END_VAR
GVL_InstruTestUIVars.g_curTestCycles:=m_testCycles;
instruTestMode(i_slaveArm);
(*
IF ABS( m_targetGripAngLast-m_targetGripAng)>0.0001  THEN
  IF  m_targetGripAngLast-m_targetGripAng<0.0001   THEN
	  m_targetGripAng:=m_targetGripAng+m_openAngleInitCompensation*g_deg2rad;
  ELSE
	  m_targetGripAng:=m_targetGripAng;
  END_IF                       
END_IF
m_targetGripAngLast:=m_targetGripAng;
*)
//TIME
fbTime.timer(bStart:=TRUE,uiTimeHour=>GVL_InstruTestUIVars.g_testTimeHour,
						  uiTimeMinute=>GVL_InstruTestUIVars.g_testTimeMinute,
						  uiTimeSecond=>GVL_InstruTestUIVars.g_testTimeSecond);
// run OTG
FOR i:=1 TO 3  DO
	m_DHJntOTG[i].run(m_targetDHJntPos[i],0.0, o_cmdAcc=>,o_cmdVel=>m_cmdDHJntVel[i],o_cmdPos=> m_cmdDHJntPos[i+3]);
END_FOR
m_gripAngleOTG.run(m_targetGripAng,0.0, o_cmdAcc=>,o_cmdVel=>,o_cmdPos=>m_cmdGripAng);

// calculate target motor joint position from DH joint position
i_slaveArm.instrument.instruIK(m_cmdDHJntPos,m_cmdGripAng, o_jntPos=>m_cmdJntPos);

// command velocity
vecSub(m_cmdJntPos, m_lastCmdJntPos, m_cmdJntVel);
vecSelfMultiNum(m_cmdJntVel, g_slaveArmCtrlFreq);
m_lastCmdJntPos:=m_cmdJntPos;
END_METHOD

// override this function in each exact controller
METHOD PROTECTED calcCmdJntTrq : BOOL
VAR_IN_OUT CONSTANT
	i_endoscopePose : ST_Frame;
	i_masterStatus :ST_MasterStatus;
	i_setupStatus: ST_SetupStatus;
	i_slaveArm :FB_SlaveArm;
END_VAR

VAR 
	nullspaceMat :Mat7d;
	ctrlTrq : Vec7d;
	i : int ;
END_VAR
// set joint torque to zero in default
m_cmdJntTrq := g_zeroVec8d;

// instrument joint control
FOR i:=1 TO 5 DO 
	m_instruCmdJntPos[i]:=m_cmdJntPos[i+3];
	m_instruCmdJntVel[i]:=m_cmdJntVel[i+3];
END_FOR

IF i_slaveArm.instrument.instruType = InstruType_UltrasoundKnifeS OR i_slaveArm.instrument.instruType = InstruType_UltrasoundKnifeU THEN
	m_usKnifeController.run(m_instruCmdJntPos,m_instruCmdJntVel, m_targetGripForceLevel, i_slaveArm, o_cmdJntTrq=>m_instruCmdJntTrq);
ELSE
	m_instruController.run(m_instruCmdJntPos,m_instruCmdJntVel, m_cmdDHJntPos[6], m_cmdDHJntVel[6], m_targetGripForceLevel, i_slaveArm, o_cmdJntTrq=>m_instruCmdJntTrq);
END_IF

FOR i:=1 TO 5 DO
	m_cmdJntTrq[i+3]:=m_instruCmdJntTrq[i];
END_FOR
END_METHOD

METHOD PUBLIC init : BOOL
VAR_IN_OUT CONSTANT
	i_slaveArm	:FB_SlaveArm;
END_VAR
VAR_IN_OUT 
	r_slaveArmCtrlCmd :ST_SlaveArmCtrlCmds;
END_VAR

VAR
	i:int;
END_VAR
SUPER^.Init(i_slaveArm,r_slaveArmCtrlCmd);
m_lastCmdJntPos:=m_cmdJntPos;
m_jntOPMode[1] := DriverOPMode_PosTrq;
m_jntOPMode[2] := DriverOPMode_PosTrq;
m_jntOPMode[3] := DriverOPMode_PosTrq;
m_jntOPMode[4] := DriverOPMode_Trq;
m_jntOPMode[5] := DriverOPMode_Trq;
m_jntOPMode[6] := DriverOPMode_Trq;
m_jntOPMode[7] := DriverOPMode_Trq;
m_jntOPMode[8] := DriverOPMode_Trq;
m_armIdx:=i_slaveArm.armIdx;
fbTime.init();

//IF i_slaveArm.instrument.onChipData.m_InstruReadSucceed AND (InstruType_UltrasoundKnifeS = i_slaveArm.instrument.m_instruType 
 //  OR InstruType_UltrasoundKnifeU = i_slaveArm.instrument.m_instruType) THEN
    m_openAngleInitCompensation:=0;
	m_instruTestMode := 0;//GVL_InstruTestUIVars.g_testMode;
//ELSE
//	m_openAngleInitCompensation:=GVL_InstruTestUIVars.g_openAngleInitCompensation;
//	m_instruTestMode := GVL_InstruTestUIVars.g_testMode+10;
//END_IF
m_testStep := 0;
m_testCycles := 1;
m_cmdDHJntPos :=i_slaveArm.curDHJntPos;
m_cmdDHJntVel :=g_zeroVec6d;
m_targetGripAng := i_slaveArm.curGripAngle;
m_targetDHJntPos[1] := i_slaveArm.curDHJntPos[4];
m_targetDHJntPos[2] := i_slaveArm.curDHJntPos[5];
m_targetDHJntPos[3] := i_slaveArm.curDHJntPos[6];

// init instrument controller
m_instruController.init(i_slaveArm,m_maxGripCurrent,m_maxGripCtrlCurrent);
m_usKnifeController.init(i_slaveArm);
m_instruType := i_slaveArm.instrument.instruType;

FOR i:=1 TO 3  DO
	m_DHJntOTG[i].init(m_cmdDHJntPos[i+3], 0, m_maxJntVel[i], m_maxJntAcc[i], g_slaveArmCtrlCycleTime);
END_FOR

m_gripAngleOTG.init(m_targetGripAng, 0, m_maxJntVel[1], m_maxJntAcc[1], g_slaveArmCtrlCycleTime);
// update commands to arm
copyCmds(r_slaveArmCtrlCmd);


iStep:=5;
END_METHOD

PROPERTY InstruBacklash : Vec5d
GET
IF m_instruType = InstruType_UltrasoundKnifeS OR m_instruType = InstruType_UltrasoundKnifeU THEN
	instruBacklash := g_zeroVec5d;
ELSE
	instruBacklash := m_instruController.m_jntBacklash;
END_IF
END_GET
END_PROPERTY

METHOD instruTestMode : BOOL
VAR_IN_OUT CONSTANT
	i_slaveArm :FB_SlaveArm;
END_VAR
VAR
	i:INT;
END_VAR
CASE m_instruTestMode OF
	0:
		m_testStep := LIMIT(0,m_testStep, 12);
		m_instruPos:=m_postureTest;
		iStep1:=12;
		iStep2:=10;
	1:
		m_testStep := LIMIT(0,m_testStep, 8);
		m_instruPos:=m_openCloseTest;
		iStep1:=7;
		iStep2:=6;
	2:
		m_testStep := LIMIT(0,m_testStep, 59);
		m_instruPos:=m_openGripMoveTest;
		iStep1:=58;
		iStep2:=57;
	3:
		m_testStep := LIMIT(0,m_testStep, 59);
		m_instruPos:=m_openGripMoveTest;
		iStep1:=58;
		iStep2:=57;
	4:
		m_testStep := LIMIT(0,m_testStep, 28);
		m_instruPos:=m_openGripMoveTest;
		iStep1:=27;
		iStep2:=26;
	5:
		m_testStep := LIMIT(0,m_testStep, 25);
		m_instruPos:=m_openGripMoveTest;
		iStep1:=24;
		iStep2:=23;
	ELSE
		RETURN;
END_CASE
bstepMove:=TRUE;
IF iStep=15 OR iStep=0 THEN 
	GVL_InstruTestUIVars.g_inPos:=1;
ELSE
	GVL_InstruTestUIVars.g_inPos:=0;	
END_IF
GVL_InstruTestUIVars.m_postureTestStep:=m_testStep+1;
CASE iStep OF
	0:;
	5:  
		FOR i:=1 TO 3 BY 1 DO
			m_targetDHJntPos[i] := m_instruPos[m_testStep+1, i]*g_deg2rad;
		END_FOR
		m_targetGripAng := m_instruPos[m_testStep+1, 4]*g_deg2rad;
		m_targetGripForceLevel:=m_instruPos[m_testStep+1, 5];
		bstepMove:=FALSE;
		iStep:=10;
	10: 
		IF ABS(m_cmdDHJntPos[4]-m_targetDHJntPos[1])< g_jntCtrlAngTolLow 
		AND ABS(m_cmdDHJntPos[5]-m_targetDHJntPos[2])< g_jntCtrlAngTolLow 	
		AND ABS(m_cmdDHJntPos[6]-m_targetDHJntPos[3])< g_jntCtrlAngTolLow 
		AND ABS(m_cmdGripAng- m_targetGripAng)< g_jntCtrlAngTolLow 
		AND bstepMove  THEN
		    iStep:=15;
	    END_IF
	15: 
		IF  GVL_InstruTestUIVars.g_nextStep THEN
			m_testStep :=m_testStep + 1;
			iStep:=20;
		ELSIF  GVL_InstruTestUIVars.g_lastStep THEN
			IF m_testStep>=1 THEN
				m_testStep :=m_testStep - 1;
			ELSE
				IF m_testCycles>1 THEN
					m_testCycles:=m_testCycles-1	;
					m_testStep:=iStep1-1;
				END_IF
			END_IF
			iStep:=20;
		END_IF
		GVL_InstruTestUIVars.g_nextStep:=FALSE;
		GVL_InstruTestUIVars.g_lastStep:=FALSE;
	20:
		iStep:=5;
		IF m_testStep =iStep1 THEN
			m_testCycles:=m_testCycles+1;
			m_testStep := 0;
		END_IF

		IF m_testCycles>=2 THEN
			m_testCycles:=m_testCycles-1;
			iStep:=25;
		END_IF

	25: 
	    m_testStep:=iStep2+1;
		FOR i:=1 TO 3 BY 1 DO
			m_targetDHJntPos[i] := m_instruPos[m_testStep+1, i]*g_deg2rad;
		END_FOR
        m_targetGripAng := m_instruPos[m_testStep+1, 4]*g_deg2rad;
        m_targetGripForceLevel:=m_instruPos[m_testStep+1, 5];
		m_testStep:=iStep2+2;
		iStep:=30;
	
    30: IF ABS(m_cmdDHJntPos[4]-m_targetDHJntPos[1])< g_jntCtrlAngTolLow 
		AND ABS(m_cmdDHJntPos[5]-m_targetDHJntPos[2])< g_jntCtrlAngTolLow 
		AND ABS(m_cmdDHJntPos[6]-m_targetDHJntPos[3])< g_jntCtrlAngTolLow 
		AND ABS(m_cmdGripAng- m_targetGripAng)< g_jntCtrlAngTolLow THEN
		    iStep:=35;
	    END_IF
	35: 
	    m_isFinished := TRUE;
		iStep:=0;
END_CASE
END_METHOD

END_FUNCTION_BLOCK

// ---- FBs_SlaveControllers/FB_SlaveCtrlFrictionTest.TcPOU
// Brief: Slave Arm test
FUNCTION_BLOCK PUBLIC FB_SlaveCtrlFrictionTest EXTENDS FB_SlaveArmCtrlBase
VAR_INPUT
END_VAR
VAR_OUTPUT
END_VAR
VAR	
	m_jntOTG:ARRAY[1..6] OF FB_secOrdTrajFilter;
	m_testStep :INT:=0;
	m_cmdDHJntPos,m_targetDHJntPos :Vec6d;
	m_cmdDHJntAcc:Vec6d;
	m_cmdGripAng:LREAL:=0;
	m_lastCmdJntPos :Vec8d ;
	m_reachTargetPos:BOOL;
	m_currentRatioMotor2Jnt:LREAL;
	m_currentLoad1:LREAL := 50;
	m_currentLoad2:LREAL := 200;
	m_trqLoad1, m_trqLoad2 :LREAL;
	m_jntFrictionNum:Vec4d;
	
	m_jntFrictionNoLoad :Vec4d;
	m_jntFrictionWithLoad:Vec4d; 

	

	
//####################################################################

END_VAR

METHOD PROTECTED calcCmdJntPos : BOOL
VAR_IN_OUT CONSTANT
	i_endoscopePose : ST_Frame;
	i_masterStatus :ST_MasterStatus;
	i_setupStatus: ST_SetupStatus;
	i_slaveArm :FB_SlaveArm;
END_VAR

VAR 
	i:INT :=0;
	angErr:Vec6d;
	errThres :LREAL;
	jntVel:Vec8d;
	jntPos:Vec6d;
END_VAR
IF m_testStep > 8 THEN 
	m_isFinished := TRUE;
END_IF

m_jntOPMode := g_slaveAllPosTrqMode; 
m_cmdJntTrq :=g_zeroVec8d;
jntVel:=i_slaveArm.curJntVel;
jntPos:=i_slaveArm.curDHJntPos;
CASE m_testStep OF 
	0: // move to start posture
		m_targetDHJntPos[4]:=pi;
		m_targetDHJntPos[5]:=-PI/2;
		m_targetDHJntPos[6]:=-80*g_deg2rad;
	1: // yaw friction without load
		m_targetDHJntPos[4]:=pi;
		m_targetDHJntPos[5]:=-PI/2;
		m_targetDHJntPos[6]:=80*g_deg2rad;
		
		IF ABS(m_cmdDHJntAcc[6])<g_smallNum THEN
			m_jntFrictionNoLoad[1]:= (m_jntFrictionNoLoad[1]*m_jntFrictionNum[1]+ABS(i_slaveArm.filtJntCurrent[4]))/(m_jntFrictionNum[1]+1);
			m_jntFrictionNum[1]:=m_jntFrictionNum[1]+1;
			
			m_jntFrictionNoLoad[2]:= (m_jntFrictionNoLoad[2]*m_jntFrictionNum[2]+ABS(i_slaveArm.filtJntCurrent[5]))/(m_jntFrictionNum[2]+1);
			m_jntFrictionNum[2]:=m_jntFrictionNum[2]+1;
		END_IF
	2: // yaw finger1  friction with load 
		m_targetDHJntPos[4]:=pi;
		m_targetDHJntPos[5]:=-PI/2;
		m_targetDHJntPos[6]:=-80*g_deg2rad;
		m_jntOPMode[4]:= DriverOPMode_Trq;
		m_cmdJntTrq[4]:= m_trqLoad1;
		
		IF ABS(m_cmdDHJntAcc[6])<g_smallNum THEN
			m_jntFrictionWithLoad[2]:= (m_jntFrictionWithLoad[2]*m_jntFrictionNum[2]+ABS(i_slaveArm.filtJntCurrent[5]))/(m_jntFrictionNum[2]+1);
			m_jntFrictionNum[2]:=m_jntFrictionNum[2]+1;
		END_IF
	3: // yaw finger2  friction with load 
		m_targetDHJntPos[4]:=pi;
		m_targetDHJntPos[5]:=-PI/2;
		m_targetDHJntPos[6]:=80*g_deg2rad;
		m_jntOPMode[5]:= DriverOPMode_Trq;
		m_cmdJntTrq[5]:= m_trqLoad1;
		
		IF ABS(m_cmdDHJntAcc[6])<g_smallNum THEN
			m_jntFrictionWithLoad[1]:= (m_jntFrictionWithLoad[1]*m_jntFrictionNum[1]+ABS(i_slaveArm.filtJntCurrent[4]))/(m_jntFrictionNum[1]+1);
			m_jntFrictionNum[1]:=m_jntFrictionNum[1]+1;
		END_IF
		
	4: // pitch  friction without load 
		m_targetDHJntPos[4]:=pi;
		m_targetDHJntPos[5]:=-PI/2+75*g_deg2Rad;
		m_targetDHJntPos[6]:=0*g_deg2rad;
	5: 
		m_targetDHJntPos[4]:=pi;
		m_targetDHJntPos[5]:=-PI/2-75*g_deg2Rad;
		m_targetDHJntPos[6]:=0*g_deg2rad;
		
		IF ABS(m_cmdDHJntAcc[5])<g_smallNum THEN
			m_jntFrictionNoLoad[3]:= (m_jntFrictionNoLoad[3]*m_jntFrictionNum[3]+ABS(i_slaveArm.filtJntCurrent[6]))/(m_jntFrictionNum[3]+1);
			m_jntFrictionNum[3]:=m_jntFrictionNum[3]+1;
		END_IF
		
	6: // pitch  friction with load 
		m_targetDHJntPos[4]:=pi;
		m_targetDHJntPos[5]:=-PI/2+75*g_deg2Rad;
		m_targetDHJntPos[6]:=0*g_deg2rad;
		m_jntOPMode[4]:= DriverOPMode_Trq;
		m_cmdJntTrq[4]:= m_trqLoad2;
		m_jntOPMode[5]:= DriverOPMode_Trq;
		m_cmdJntTrq[5]:= m_trqLoad2;
		
		IF ABS(m_cmdDHJntAcc[5])<g_smallNum THEN
			m_jntFrictionWithLoad[3]:= (m_jntFrictionWithLoad[3]*m_jntFrictionNum[3]+ABS(i_slaveArm.filtJntCurrent[6]))/(m_jntFrictionNum[3]+1);
			m_jntFrictionNum[3]:=m_jntFrictionNum[3]+1;
		END_IF
	7: // roll friction without load 
		m_targetDHJntPos[4]:=-pi;
		m_targetDHJntPos[5]:=-PI/2+75*g_deg2Rad;
		m_targetDHJntPos[6]:=0*g_deg2rad;
		IF ABS(m_cmdDHJntAcc[4])<g_smallNum THEN
			m_jntFrictionNoLoad[4]:= (m_jntFrictionNoLoad[4]*m_jntFrictionNum[4]+ABS(i_slaveArm.filtJntCurrent[7]))/(m_jntFrictionNum[4]+1);
			m_jntFrictionNum[4]:=m_jntFrictionNum[4]+1;
		END_IF
	8: 
		m_targetDHJntPos[4]:=-pi;
		m_targetDHJntPos[5]:=-PI/2;
		m_targetDHJntPos[6]:=0*g_deg2rad;
		
END_CASE

// check if finish current motion
vecSub(m_cmdDHJntPos, m_targetDHJntPos, angErr);
IF norm(angErr)< 1*g_deg2Rad AND norm(jntVel)<1*g_deg2Rad THEN
	m_testStep := m_testStep+1;
	m_jntFrictionNum:=g_zeroVec4d;
END_IF


FOR i:=4 TO 6 DO 
	m_jntOTG[i].run(m_targetDHJntPos[i],0.0, o_cmdAcc=>m_cmdDHJntAcc[i],o_cmdVel=>,o_cmdPos=> m_cmdDHJntPos[i]);
END_FOR

i_slaveArm.instrument.instruIK(m_cmdDHJntPos,m_cmdGripAng, o_jntPos=>m_cmdJntPos);

// command velocity
vecSub(m_cmdJntPos, m_lastCmdJntPos, m_cmdJntVel);
vecSelfMultiNum(m_cmdJntVel, g_slaveArmCtrlFreq);
m_lastCmdJntPos:=m_cmdJntPos;
END_METHOD

// override this function in each exact controller
METHOD PROTECTED calcCmdJntTrq : BOOL
VAR_IN_OUT CONSTANT
	i_endoscopePose : ST_Frame;
	i_masterStatus :ST_MasterStatus;
	i_setupStatus: ST_SetupStatus;
	i_slaveArm :FB_SlaveArm;
END_VAR

VAR 
	nullspaceMat :Mat7d;
	ctrlTrq : Vec7d;
	i : int ;
END_VAR
END_METHOD

METHOD PUBLIC init : BOOL
VAR_IN_OUT CONSTANT
	i_slaveArm	:FB_SlaveArm;
END_VAR
VAR_IN_OUT 
	r_slaveArmCtrlCmd :ST_SlaveArmCtrlCmds;
END_VAR

VAR
	i:int;
END_VAR
SUPER^.Init(i_slaveArm,r_slaveArmCtrlCmd);
m_lastCmdJntPos:=m_cmdJntPos;
m_jntOPMode := g_slaveAllPosTrqMode; 

m_testStep:=0;
m_cmdDHJntPos :=i_slaveArm.curDHJntPos;
m_targetDHJntPos:=m_cmdDHJntPos;
m_cmdGripAng:=0;
m_lastCmdJntPos:=m_cmdJntPos;
m_reachTargetPos:=FALSE;

m_currentRatioMotor2Jnt:=GVL_SlaveMotorParameters.g_motorTrqConst[4]*GVL_SlaveMotorParameters.g_motorReduction[4]/1000;
m_trqLoad1 := m_currentLoad1 * m_currentRatioMotor2Jnt;
m_trqLoad2 := m_currentLoad2 * m_currentRatioMotor2Jnt;


FOR i:=1 TO 6  DO
	m_jntOTG[i].init(m_cmdDHJntPos[i], 0, 10*g_deg2Rad, 4, g_slaveArmCtrlCycleTime);
END_FOR

m_jntFrictionNoLoad:=g_zeroVec4d;
m_jntFrictionWithLoad:=g_zeroVec4d;
m_jntFrictionNum:=g_zeroVec4d;

// update commands to arm
copyCmds(r_slaveArmCtrlCmd);
END_METHOD

END_FUNCTION_BLOCK

// ---- FBs_SlaveControllers/FB_SlaveCtrMotorGoHome.TcPOU
// Brief: Mounting Panel
FUNCTION_BLOCK PUBLIC FB_SlaveCtrMotorGoHome EXTENDS FB_SlaveArmCtrlBase
VAR
	// motorGoHomeStatus
	m_motorGoHomeStatus :INT := 0;
	
	// mount motion planning
	m_jntOTG :ARRAY[1..5] OF FB_secOrdTrajFilter;
	m_motorGoHomeVel :LREAL := 2*pi;
	m_motorGoHomeAcc :LREAL := 4*pi;
	m_targetHomePos :Vec5d;
END_VAR

// override this function in each exact controller
METHOD PROTECTED calcCmdJntPos : BOOL
VAR_IN_OUT CONSTANT
	i_endoscopePose : ST_Frame;
	i_masterStatus :ST_MasterStatus;
	i_setupStatus: ST_SetupStatus;
	i_slaveArm :FB_SlaveArm;
END_VAR

VAR 
	i :INT;
	curJntPos :Vec8d;
	cycleNum :LREAL;
END_VAR

curJntPos := i_slaveArm.curJntPos;

CASE m_motorGoHomeStatus OF
	
	// determine zero position 
	0:
		FOR i:=1 TO 5 DO
			cycleNum := FLOOR(curJntPos[i+3]/g_2pi);
			m_targetHomePos[i]:=cycleNum* g_2Pi;
		END_FOR
		m_motorGoHomeStatus :=1;
	
	// move back to zero position
	1:
		m_isFinished:=TRUE;
		FOR i:=1 TO 5 DO
			IF ABS(m_targetHomePos[i]-curJntPos[i+3])>GVL_SlaveControlParameters.g_jntCtrlAngTolHigh THEN
				m_isFinished:=FALSE;
				EXIT;
			END_IF
		END_FOR
END_CASE


FOR i:=1 TO 5 DO
	m_jntOTG[i].run(m_targetHomePos[i],0.0, o_cmdAcc=>m_cmdJntAcc[3+i],o_cmdVel=>m_cmdJntVel[3+i],o_cmdPos=>m_cmdJntPos[i+3]);
END_FOR
END_METHOD

METHOD PUBLIC init : BOOL
VAR_IN_OUT CONSTANT
	i_slaveArm	:FB_SlaveArm;
END_VAR
VAR_IN_OUT 
	r_slaveArmCtrlCmd :ST_SlaveArmCtrlCmds;
END_VAR
VAR
	i : INT;
END_VAR
SUPER^.Init(i_slaveArm,r_slaveArmCtrlCmd);//T
m_jntOPMode[4] := DriverOPMode_Pos;
m_jntOPMode[5] := DriverOPMode_Pos;
m_jntOPMode[6] := DriverOPMode_Pos;
m_jntOPMode[7] := DriverOPMode_Pos;
m_jntOPMode[8] := DriverOPMode_Pos;

m_motorGoHomeStatus:=0;
FOR i:=1 TO 5 DO
	m_targetHomePos[i]:=m_cmdJntPos[i+3];
	m_jntOTG[i].init(m_targetHomePos[i], 0,m_motorGoHomeVel, m_motorGoHomeAcc, g_slaveArmCtrlCycleTime);
END_FOR

// update commands to arm
copyCmds(r_slaveArmCtrlCmd);
END_METHOD

END_FUNCTION_BLOCK

// ---- FBs_Robots/FB_SlaveRobot.TcPOU
FUNCTION_BLOCK FB_SlaveRobot
VAR
	// slave arms, responsible for arm kinematic and control
	m_slaveArms :ARRAY[1..g_sArmNum] OF FB_SlaveArm;
	
	// arm light control word
	m_lightCrlWord :ARRAY [1..4] OF UDINT;
	
	// arm state
	m_slaveArmState:ARRAY[1..g_sArmNum] OF E_SlaveArmState:=[g_sArmNum(E_SlaveArmState.SlaveArmState_Error)];
	m_lastSlaveArmState:ARRAY[1..g_sArmNum] OF E_SlaveArmState:=[g_sArmNum(E_SlaveArmState.SlaveArmState_Error)];
	m_nextSlaveArmState:ARRAY[1..g_sArmNum] OF E_SlaveArmState:=[g_sArmNum(E_SlaveArmState.SlaveArmState_Error)];
	
	// flag if panel and instrument mounted
	m_panelMountedFlag :ARRAY[1..g_sArmNum] OF BOOL :=[g_sArmNum(FALSE)];
	m_instrumentMountedFlag :ARRAY[1..g_sArmNum] OF BOOL :=[g_sArmNum(FALSE)];
	
	// all arm controller instance 
	m_armCtrlFactory :ARRAY[1..g_sArmNum,1..SlaveArmState_totalNum] OF I_SlaveArmCtrl;
	m_armError :ARRAY[1..g_sArmNum] OF FB_SlaveCtrlError;
	m_armInit :ARRAY[1..g_sArmNum] OF FB_SlaveCtrlInit;
	m_armSelfCheck :ARRAY[1..g_sArmNum] OF FB_SlaveCtrlSelfCheck;
	m_armStandBy :ARRAY[1..g_sArmNum] OF FB_SlaveCtrlStandBy;
	m_mountPanel :ARRAY[1..g_sArmNum] OF FB_SlaveCtrlMountPanel;
	m_panelReady :ARRAY[1..g_sArmNum] OF FB_SlaveCtrlPanelReady;
	m_mountInstru :ARRAY[1..g_sArmNum] OF FB_SlaveCtrlMountInstru;
	m_instruReady :ARRAY[1..g_sArmNum] OF FB_SlaveCtrlInstruReady;
	m_armMasterSlave :ARRAY[1..g_sArmNum] OF FB_SlaveCtrlMasterSlave;
	m_scopeReady :ARRAY[1..g_sArmNum] OF FB_SlaveCtrlScopeReady;
	m_armEndoscope :ARRAY[1..g_sArmNum] OF FB_SlaveCtrlEndoscope;
	m_armAdjust :ARRAY[1..g_sArmNum] OF FB_SlaveCtrlAdjust;
	m_armPackage :ARRAY[1..g_sArmNum] OF FB_SlaveCtrlPackage;
	m_armCart :ARRAY[1..g_sArmNum] OF FB_SlaveCtrlCart;
	m_armGraCali :ARRAY[1..g_sArmNum] OF FB_SlaveCtrlGraCali;
	m_armTest :ARRAY[1..g_sArmNum] OF FB_SlaveCtrlTest;
	m_instruRetract :ARRAY[1..g_sArmNum] OF FB_SlaveCtrlInstruRetract;
	m_instruInvasion :ARRAY[1..g_sArmNum] OF FB_SlaveCtrlInstruInvasion;
	m_armDisable :ARRAY[1..g_sArmNum] OF FB_SlaveCtrlDisable;
	m_instruCali :ARRAY[1..g_sArmNum] OF FB_SlaveCtrlInstruCali;
	m_scopeToggle :ARRAY[1..g_sArmNum] OF FB_SlaveCtrlScopeToggle;
	m_Performance :ARRAY[1..g_sArmNum] OF FB_SlaveCtrlPerformance;
	m_armStop :ARRAY[1..g_sArmNum] OF FB_SlaveCtrlStop;
	m_instruAutoTest :ARRAY[1..g_sArmNum] OF FB_SlaveCtrlInstruAutoTest;
	m_instruManualTest :ARRAY[1..g_sArmNum] OF FB_SlaveCtrlInstruManualTest;
	m_instruVerify :ARRAY[1..g_sArmNum] OF FB_SlaveCtrlInstruVerify;
	m_frictionTest :ARRAY[1..g_sArmNum] OF FB_SlaveCtrlFrictionTest;
	
	// arm controller interface
	m_armCtrl :ARRAY[1..g_sArmNum] OF I_SlaveArmCtrl;
	m_armCtrlCmds :ARRAY[1..g_sArmNum] OF ST_SlaveArmCtrlCmds;
	m_motorGoHome: ARRAY[1..g_sArmNum] OF FB_SlaveCtrMotorGoHome;
	m_powerBoxCalibration: ARRAY[1..g_sArmNum] OF FB_SlaveCtrlPowerBoxCalibration;
	fbTonMotorGoHomeState: TON;
	fbTonPowerBoxCalibrationState: TON;
	m_endoscopeTest: ARRAY[1..g_sArmNum] OF FB_SlaveCtrlInstruEndoscopeTest;
	m_enableMode:BOOL;
	
	m_frictionTestButtonRise :R_TRIG;
	m_frictionTestButtonFall :F_TRIG;
	m_frictionTestStart, m_frictionTestEnd:BOOL;
END_VAR

METHOD PROTECTED controllerTransit : BOOL
VAR_INPUT
END_VAR
VAR
	i:int;
END_VAR
FOR i:=1 TO g_sArmNum DO 
	// Controller transit
	IF m_nextSlaveArmState[i]<> m_slaveArmState[i] THEN
		// reset current controller
		m_armCtrl[i].reset();
		
		// transit to new controller
		m_lastSlaveArmState[i]:=m_slaveArmState[i];
		m_slaveArmState[i]:=m_nextSlaveArmState[i];
		m_armCtrl[i]:=m_armCtrlFactory[i,m_slaveArmState[i]];
		
		// init next controller
		m_armCtrl[i].Init(m_slaveArms[i],m_armCtrlCmds[i]);
		m_slaveArms[i].updateCmds(m_armCtrlCmds[i]);
	END_IF
END_FOR
END_METHOD

METHOD PUBLIC Init : BOOL
VAR_INPUT
END_VAR
VAR
	i:INT;
END_VAR
FOR i:=1 TO g_sArmNum DO
	// arm init
	m_slaveArms[i].Init(i);
	m_slaveArmState[i]:=SlaveArmState_Init;
	m_lastSlaveArmState[i]:=SlaveArmState_Init;
	m_nextSlaveArmState[i]:=SlaveArmState_Init;
	
	// command init
	m_armCtrlCmds[i].m_jntEnableFlag := g_zeroVec8i;
	m_armCtrlCmds[i].m_jntOPMode := g_slaveAllPosMode;
	m_armCtrlCmds[i].m_cmdCartPose := m_slaveArms[i].curCartPose;
	m_armCtrlCmds[i].m_cmdCartTwist := g_zeroVec6d;
	m_armCtrlCmds[i].m_cmdJntPos := m_slaveArms[i].curJntPos;
	m_armCtrlCmds[i].m_cmdJntVel := g_zeroVec8d;
	m_armCtrlCmds[i].m_cmdJntAcc := g_zeroVec8d;
	m_armCtrlCmds[i].m_cmdJntTrq := g_zeroVec8d;
	
	// generate controller factory
	m_armCtrlFactory[i,SlaveArmState_Error] := m_armError[i];
	m_armCtrlFactory[i,SlaveArmState_Init] := m_armInit[i];
	m_armCtrlFactory[i,SlaveArmState_SelfCheck] := m_armSelfCheck[i];
	m_armCtrlFactory[i,SlaveArmState_Standby] := m_armStandBy[i];
	m_armCtrlFactory[i,SlaveArmState_MountPanel] := m_mountPanel[i];
	m_armCtrlFactory[i,SlaveArmState_PanelReady] := m_panelReady[i];
	m_armCtrlFactory[i,SlaveArmState_MountInstru] := m_mountInstru[i];
	m_armCtrlFactory[i,SlaveArmState_InstruReady] := m_instruReady[i];
	m_armCtrlFactory[i,SlaveArmState_MasterSlave] := m_armMasterSlave[i];
	m_armCtrlFactory[i,SlaveArmState_ScopeReady] := m_scopeReady[i];
	m_armCtrlFactory[i,SlaveArmState_EndoScope] := m_armEndoscope[i];
	m_armCtrlFactory[i,SlaveArmState_Adjust] := m_armAdjust[i];
	m_armCtrlFactory[i,SlaveArmState_Package] := m_armPackage[i];
	m_armCtrlFactory[i,SlaveArmState_Cart] := m_armCart[i];
	m_armCtrlFactory[i,SlaveArmState_GravityCali] := m_armGraCali[i];
	m_armCtrlFactory[i,SlaveArmState_Test] := m_armTest[i];
	m_armCtrlFactory[i,SlaveArmState_InstruRetract] := m_instruRetract[i];
	m_armCtrlFactory[i,SlaveArmState_InstruInvasion] := m_instruInvasion[i];
	m_armCtrlFactory[i,SlaveArmState_Disable] := m_armDisable[i];
	m_armCtrlFactory[i,SlaveArmState_InstruCali] := m_instruCali[i];
	m_armCtrlFactory[i,SlaveArmState_ScopeToggle] := m_scopeToggle[i];
	m_armCtrlFactory[i,SlaveArmState_Performance] := m_Performance[i];
	m_armCtrlFactory[i,SlaveArmState_Stop] := m_armStop[i];
	m_armCtrlFactory[i,SlaveArmState_InstruAutoTest] := m_instruAutoTest[i];
	m_armCtrlFactory[i,SlaveArmState_InstruManualTest] := m_instruManualTest[i];
	m_armCtrlFactory[i,SlaveArmState_InstruVerify] := m_instruVerify[i];
	m_armCtrlFactory[i,SlaveArmState_MotorGoHome] := m_motorGoHome[i];
	m_armCtrlFactory[i,SlaveArmState_PowerBoxCalibration] := m_powerBoxCalibration[i];
	m_armCtrlFactory[i,SlaveArmState_EndoscopeTest] := m_endoscopeTest[i];
	m_armCtrlFactory[i,SlaveArmState_FrictionTest] := m_frictionTest[i];
	// assign controller
	m_armCtrl[i]:=m_armCtrlFactory[i,m_slaveArmState[i]];
	m_armCtrl[i].Init(m_slaveArms[i],m_armCtrlCmds[i]);
END_FOR
END_METHOD

METHOD PUBLIC run : BOOL
VAR_IN_OUT CONSTANT
	i_slaveInputDataPool:ST_SlaveInputDataPool;
END_VAR
VAR
	i:INT;
	nullScopePose :ST_Frame;
	nullSetupStatus:ST_SetupStatus;
	nullMasterStatus:ST_MasterStatus;
	
	
END_VAR
FOR i:=1 TO g_sArmNum DO
	// update dynamic data
	m_slaveArms[i].updateDyna(i_slaveInputDataPool.m_slaveDynaData);
								
	// update slave arm kinematics
	m_slaveArms[i].updateStatus();
END_FOR

//update arm light
updateArmLight(i_slaveInputDataPool);

// state machine transition
stateMachine(i_slaveInputDataPool);

// controller transition
controllerTransit();

FOR i:=1 TO g_sArmNum DO
	// null ptr check
	ASSERT(0 <> m_armCtrl[i]);
	
	// run controller
	m_armCtrl[i].run(nullScopePose, nullMasterStatus, nullSetupStatus,m_SlaveArms[i],m_armCtrlCmds[i]);

	// update commands to drivers
	m_slaveArms[i].updateCmds(m_armCtrlCmds[i]);

END_FOR
// ################# update insrument UI data #########################################
FOR i:=1 TO 5 DO 
	GVL_InstruTestUIVars.g_curInstruJntPos[i]:= m_slaveArms[1].curJntPos[i+3];
	GVL_InstruTestUIVars.g_curInstruJntCurrent[i]:= m_slaveArms[1].filtJntCurrent[i+3];
	GVL_InstruTestUIVars.g_instruZeroPos[i]:= m_slaveArms[1].instrument.onChipData.m_InstruPos[i];
END_FOR

FOR i:=1 TO 3 DO
		GVL_InstruTestUIVars.g_curInstruDHPos[i]:= m_slaveArms[1].curDHJntPos[i+3];
END_FOR

GVL_InstruTestUIVars.g_curGripAng := m_slaveArms[1].curGripAngle;
GVL_InstruTestUIVars.g_enabled := m_slaveArms[1].m_joints[6].isEnabled() ;

m_frictionTestButtonRise(CLK:=GVL_InstruTestUIVars.g_instruFrictionTest,  Q=>m_frictionTestStart);
m_frictionTestButtonFall(CLK:=GVL_InstruTestUIVars.g_instruFrictionTest,  Q=>m_frictionTestEnd);
END_METHOD

// state machine check and transit 
METHOD PROTECTED stateMachine : BOOL
VAR_IN_OUT CONSTANT
		i_slavesInputDataPool:ST_SlaveInputDataPool;
END_VAR
VAR
	i,j:INT;
END_VAR
// check instrument state
FOR i:=1 TO g_sArmNum DO
	// statues check
	IF m_slaveArms[i].panelOn = FALSE THEN
		m_panelMountedFlag[i]:=FALSE;
	END_IF
	IF m_slaveArms[i].instruOn = FALSE THEN
		m_instrumentMountedFlag[i]:=FALSE;
	END_IF
END_FOR

// state machine transit
FOR i:=1 TO g_sArmNum DO
	CASE m_slaveArmState[i] OF
		// init
		SlaveArmState_Init:
			m_slaveArms[i].instrument.resetArmLED :=TRUE;
			// to standby
			IF m_armCtrl[i].isFinished  THEN
				m_nextSlaveArmState[i]:=SlaveArmState_Standby;
			END_IF
		
		//standby
		SlaveArmState_Standby:
			// to mount panel
			IF m_slaveArms[i].panelOn AND ((GVL_InstruTestUIVars.g_snappingSeparator AND NOT m_slaveArms[i].instruOn) OR  m_panelMountedFlag[i] )AND NOT GVL_InstruTestUIVars.g_powerBoxCalibration THEN 
				IF m_panelMountedFlag[i] THEN
					m_nextSlaveArmState[i]:=SlaveArmState_PanelReady;
				ELSE
					m_nextSlaveArmState[i]:=SlaveArmState_MountPanel;
				END_IF
			ELSIF GVL_InstruTestUIVars.g_goHome AND NOT m_slaveArms[i].instruOn THEN  
				GVL_InstruTestUIVars.g_beHomed:=FALSE;
				m_nextSlaveArmState[i]:=SlaveArmState_MotorGoHome;
			END_IF
			IF GVL_InstruTestUIVars.g_powerBoxCalibration THEN
				GVL_InstruTestUIVars.g_powerBoxCalibrationed:=FALSE;;
				IF m_slaveArms[i].panelOn THEN 
					m_nextSlaveArmState[i]:=SlaveArmState_PowerBoxCalibration;
				END_IF
			END_IF
		SlaveArmState_MotorGoHome:
			// to Standby
			IF m_armCtrl[i]. isFinished THEN
				m_nextSlaveArmState[i]:=SlaveArmState_Standby;
				GVL_InstruTestUIVars.g_beHomed:=TRUE;
			// to standby
			ELSIF fbTonMotorGoHomeState.Q THEN
				m_nextSlaveArmState[i]:=SlaveArmState_Standby;
			END_IF
		SlaveArmState_PowerBoxCalibration:
			IF m_armCtrl[i]. isFinished THEN
				GVL_InstruTestUIVars.g_powerBoxCalibration:=FALSE;
				GVL_InstruTestUIVars.g_powerBoxCalibrationed:=TRUE;
				FOR j:=4 TO g_sJntNum DO
					GVL_InstruTestUIVars.g_powerBoxCalibrationPos[i,j]:=SlaveArmControl.m_slaveRobot.m_slaveArms[i].m_joints[j].m_motorInputs.m_linkEncoder;
				END_FOR
				GVL_SlaveJointEncoderCaliData.g_caliLinkEncoder:=GVL_InstruTestUIVars.g_powerBoxCalibrationPos;
				IF NOT m_slaveArms[i].panelOn THEN
					GVL_InstruTestUIVars.g_powerBoxCalibrationFlag:=FALSE;
					m_nextSlaveArmState[i]:=SlaveArmState_Standby;;
					m_slaveArms[i].setSaveCaliLinkEncoder();
				END_IF
			// to standby
			ELSIF fbTonPowerBoxCalibrationState.Q AND NOT m_slaveArms[i].panelOn THEN
				m_nextSlaveArmState[i]:=SlaveArmState_Standby;
			END_IF
		//mount panel
		SlaveArmState_MountPanel:
			// to panel ready
			IF m_armCtrl[i]. isFinished THEN
				m_nextSlaveArmState[i]:=SlaveArmState_PanelReady;
				m_panelMountedFlag[i] :=TRUE;
				
			// to standby
			ELSIF NOT(m_slaveArms[i].panelOn) THEN
				m_nextSlaveArmState[i]:=SlaveArmState_Standby;
			END_IF
		
		//panel ready
		SlaveArmState_PanelReady:
			// to standby
			IF NOT(m_slaveArms[i].panelOn) THEN
				m_nextSlaveArmState[i]:=SlaveArmState_Standby;
			
			// to instrument caliberation
			ELSIF GVL_InstruTestUIVars.g_instruCaliFlag THEN
				m_nextSlaveArmState[i] := SlaveArmState_InstruCali;
			ELSIF (GVL_InstruTestUIVars.g_instrumentAutoSnapping OR m_instrumentMountedFlag[i]) AND m_slaveArms[i].instruOn   THEN
				IF m_instrumentMountedFlag[i] THEN
					// to scope ready
					IF  InstruType_endoscope = m_slaveArms[i].instrument.m_instruType AND m_slaveArms[i].instruReady() THEN 
						m_nextSlaveArmState[i]:=SlaveArmState_ScopeReady;
					// to instrument ready
					ELSE
						m_nextSlaveArmState[i]:=SlaveArmState_InstruReady;
					END_IF
				// to mount instrument/endoscope
				ELSE
					m_nextSlaveArmState[i]:=SlaveArmState_MountInstru;
				END_IF
			END_IF
			
		//mount instrument
		SlaveArmState_MountInstru:
			// to panel ready
			IF NOT(m_slaveArms[i].instruOn)  THEN
				m_nextSlaveArmState[i]:=SlaveArmState_PanelReady;
			ELSIF m_armCtrl[i].isFinished THEN
				m_instrumentMountedFlag[i] :=TRUE;
				m_nextSlaveArmState[i]:=SlaveArmState_PanelReady;
				
			END_IF
		
		// instrument ready
		SlaveArmState_InstruReady:
			// to instrument standby
			IF  NOT(m_slaveArms[i].instruOn)  THEN
				m_nextSlaveArmState[i]:=SlaveArmState_Standby;
				GVL_InstruTestUIVars.g_readRFIDFlag:=FALSE;
			// to instrument caliberation
			ELSIF GVL_InstruTestUIVars.g_instruCaliFlag THEN
				m_nextSlaveArmState[i] := SlaveArmState_InstruCali;
				
			// to instrument auto test
			ELSIF GVL_InstruTestUIVars.g_instruAutoTestFlag THEN
				m_nextSlaveArmState[i] := SlaveArmState_InstruAutoTest;
				
			// to instrument manual test
			ELSIF GVL_InstruTestUIVars.g_instruManualTestFlag THEN
				m_nextSlaveArmState[i] := SlaveArmState_InstruManualTest;
				
			// to instrument verify
			ELSIF GVL_InstruTestUIVars.g_instruVerifyFlag THEN
				m_nextSlaveArmState[i] := SlaveArmState_InstruVerify;
				
			// to instrument verify
			ELSIF GVL_InstruTestUIVars.g_endoscopeTest THEN
				m_nextSlaveArmState[i] := SlaveArmState_EndoscopeTest;
				
			//to friction Test
			ELSIF m_frictionTestStart THEN
				m_nextSlaveArmState[i] := SlaveArmState_FrictionTest;
			END_IF
			
		//instrument caliberation
		SlaveArmState_InstruCali:
			// to standby
			IF  NOT(GVL_InstruTestUIVars.g_instruCaliFlag)  THEN
				m_nextSlaveArmState[i]:=SlaveArmState_Standby;
			END_IF
			
		//instrument auto test
		SlaveArmState_InstruAutoTest:
			// to stop
			IF  NOT( m_slaveArms[1].instruOn) OR NOT(GVL_InstruTestUIVars.g_instruAutoTestFlag)  THEN
				m_nextSlaveArmState[i]:=SlaveArmState_Stop;
				GVL_InstruTestUIVars.g_readRFIDFlag:=FALSE;
				m_armStop[i].setInstruBacklash(m_instruAutoTest[i].InstruBacklash);
			END_IF
			IF m_armCtrl[i].isFinished THEN
				GVL_InstruTestUIVars.g_instruAutoTestFlag:=FALSE;
			END_IF
		//instrument manual test
		SlaveArmState_InstruManualTest:
			// to stop
			IF  NOT( m_slaveArms[1].instruOn) OR NOT(GVL_InstruTestUIVars.g_instruManualTestFlag)  THEN
				m_nextSlaveArmState[i]:=SlaveArmState_Stop;
				m_armStop[i].setInstruBacklash(m_instruManualTest[i].InstruBacklash);
				GVL_InstruTestUIVars.g_readRFIDFlag:=FALSE;
			END_IF
			
		//instrument verify
		SlaveArmState_InstruVerify:
			// to stop
			IF  NOT( m_slaveArms[1].instruOn) OR NOT(GVL_InstruTestUIVars.g_instruVerifyFlag)  THEN
				m_nextSlaveArmState[i]:=SlaveArmState_Stop;
				GVL_InstruTestUIVars.g_readRFIDFlag:=FALSE;
				m_armStop[i].setInstruBacklash(m_instruVerify[i].InstruBacklash);
			END_IF
			IF m_armCtrl[i].isFinished THEN
				GVL_InstruTestUIVars.g_instruVerifyFlag:=FALSE;
			END_IF
			
		//arm stop
		SlaveArmState_Stop:
			// to standby
			IF  m_armCtrl[i].isFinished THEN
				m_nextSlaveArmState[i]:=SlaveArmState_Standby;
			END_IF
			
		SlaveArmState_Disable:
			// to init
			IF  NOT GVL_InstruTestUIVars.g_powerOn  THEN
				m_nextSlaveArmState[i]:=SlaveArmState_Init;
			END_IF
		    IF  NOT( m_slaveArms[1].instruOn) THEN
				m_nextSlaveArmState[i]:=SlaveArmState_Init;
			END_IF
			
		SlaveArmState_EndoscopeTest:
			IF  NOT( m_slaveArms[1].instruOn) OR NOT(GVL_InstruTestUIVars.g_endoscopeTest)  THEN
				m_nextSlaveArmState[i]:=SlaveArmState_Stop;
			END_IF
			
		SlaveArmState_FrictionTest:
			// to stop
			IF  NOT( m_slaveArms[1].instruOn) OR m_armCtrl[i].isFinished OR m_frictionTestEnd  THEN
				m_nextSlaveArmState[i]:=SlaveArmState_Standby;
			END_IF
	END_CASE
	IF NOT m_slaveArms[i].instruOn THEN
		GVL_InstruTestUIVars.g_instruCaliState:=FALSE;
	END_IF
	IF GVL_InstruTestUIVars.g_powerOn THEN 
		m_nextSlaveArmState[i]:=SlaveArmState_Disable;
	END_IF
	IF GVL_InstruTestUIVars.g_motorStops THEN 
		GVL_InstruTestUIVars.g_motorStops:=FALSE;
		m_nextSlaveArmState[i]:=SlaveArmState_Stop;
	END_IF
	IF m_slaveArmState[i]<>SlaveArmState_PowerBoxCalibration AND m_slaveArmState[i]<>SlaveArmState_Standby THEN
		GVL_InstruTestUIVars.g_powerBoxCalibration:=FALSE;
	END_IF
	IF m_slaveArmState[i]<>SlaveArmState_MotorGoHome AND m_slaveArmState[i]<>SlaveArmState_Standby THEN
		GVL_InstruTestUIVars.g_beHomed:=FALSE;
	END_IF
	
	
GVL_InstruTestUIVars.g_stateMachine:=m_slaveArmState[i];
	IF GVL_InstruTestUIVars.g_manualPowerBoxCalibration THEN
		FOR j:=4 TO g_sJntNum DO
			GVL_InstruTestUIVars.g_powerBoxCalibrationPos[i,j]:=SlaveArmControl.m_slaveRobot.m_slaveArms[i].m_joints[j].m_motorInputs.m_linkEncoder;
		END_FOR
		//GVL_SlaveJointEncoderCaliData.g_caliLinkEncoder:=GVL_InstruTestUIVars.g_powerBoxCalibrationPos;
		GVL_InstruTestUIVars.g_manualPowerBoxCalibration:=FALSE;
		GVL_InstruTestUIVars.g_powerBoxCalibrationFlag:=FALSE;
		m_slaveArms[i].setSaveCaliLinkEncoder();
	END_IF
END_FOR


m_enableMode:=TRUE;
GVL_InstruTestUIVars.g_logOutEnable:=GVL_InstruTestUIVars.g_stateMachine<>SlaveArmState_InstruAutoTest;
GVL_InstruTestUIVars.g_snappingSeparatoring:=GVL_InstruTestUIVars.g_stateMachine=SlaveArmState_MountPanel;
GVL_InstruTestUIVars.g_instruAutoSnapping:=GVL_InstruTestUIVars.g_stateMachine=SlaveArmState_MountInstru;
GVL_InstruTestUIVars.g_instruCalibrationing:=m_instruCali[1].getState AND GVL_InstruTestUIVars.g_stateMachine=SlaveArmState_InstruCali;
GVL_MES.g_autoTestMode:=m_instruAutoTest[1].getTestMode;
GVL_InstruTestUIVars.g_forceBipolarModeAllowed := InstruType_ForceBipolar = m_slaveArms[1].instrument.instruTypeInfo.m_InstruID;
GVL_InstruTestUIVars.g_instruFrictionTestAllowed := m_slaveArms[1].instrument.onChipData.m_InstruReadSucceed AND m_instrumentMountedFlag[1];
GVL_InstruTestUIVars.g_testEnable:=m_slaveArms[1].instrument.onChipData.m_InstruReadSucceed AND m_instrumentMountedFlag[1];
IF NOT GVL_InstruTestUIVars.g_testEnable THEN
	GVL_InstruTestUIVars.g_instruAutoTestFlag:=FALSE;
	GVL_InstruTestUIVars.g_instruManualTestFlag:=FALSE;
	GVL_InstruTestUIVars.g_instruVerifyFlag:=FALSE;
END_IF
GVL_InstruTestUIVars.g_standbyEnable:=GVL_InstruTestUIVars.g_stateMachine=SlaveArmState_Standby AND NOT m_slaveArms[1].panelOn;
END_METHOD

METHOD updateArmLight : BOOL
VAR_INPUT
	i_slaveInputDataPool:ST_SlaveInputDataPool;
END_VAR

VAR
	i : INT;
END_VAR
//*******************机械臂与动力盒上的灯光写入********************
//不可恢复性故障-----红色常亮
//可恢复故障----琥珀色-先闪烁5s、再进行常亮
//正处于器械控制或者端口控制状态-----蓝色闪烁
//该手术臂正在执行一项需要用户短时间等待的活动、例如器械卡接----蓝色-脉动闪烁
//工具更换引导正在进行中-----绿色闪烁
//未通电、已禁用、已收起----------关
//系统正常运行-----蓝色常亮
//灯光颜色--0-灯灭、1蓝灯常亮、2蓝灯闪烁、3琥珀色闪烁、4红灯闪烁、5绿灯常亮、6绿灯闪烁、7红灯常亮、8琥珀色常亮、9蓝灯脉动式闪烁

FOR i := 1 TO g_sArmNum BY 1 DO
	IF m_slaveArmState[i] = SlaveArmState_Error THEN
		m_lightCrlWord[i] := ArmLight_AmberBlink;
	ELSIF m_slaveArmState[i] = SlaveArmState_MountPanel OR m_slaveArmState[i] = SlaveArmState_MountInstru THEN
		m_lightCrlWord[i] := ArmLight_BluePulse;
	ELSIF m_slaveArmState[i] = SlaveArmState_InstruRetract OR m_slaveArmState[i] = SlaveArmState_Adjust THEN
		m_lightCrlWord[i] := ArmLight_BlueBlink;
	ELSIF m_slaveArmState[i] = SlaveArmState_InstruInvasion THEN
		m_lightCrlWord[i] := ArmLight_GreenBlink;
	ELSIF m_slaveArmState[i] = SlaveArmState_Disable THEN
		m_lightCrlWord[i] := ArmLight_Off;
	ELSE
		m_lightCrlWord[i] := ArmLight_BlueOn;
	END_IF

	m_slaveArms[i].checkLight(m_lightCrlWord[i]);
END_FOR
END_METHOD

END_FUNCTION_BLOCK

// ---- FBs_SlaveControllers/FB_SlaveCtrlInit.TcPOU
// Brief: Slave Arm Init
FUNCTION_BLOCK PUBLIC FB_SlaveCtrlInit EXTENDS FB_SlaveArmCtrlBase
VAR_INPUT
END_VAR
VAR_OUTPUT
END_VAR
VAR
	m_initState :INT :=0;
	
	// SDO writer
	m_MotorCurrentSDOWrite: ARRAY[1..5] OF FB_EcCoESdoWrite;
	// power box joint motor rated current
	m_wristJntRatedCurrent : DINT := 250;
END_VAR

// override this function in each exact controller
METHOD PROTECTED calcCmdJntPos : BOOL
VAR_IN_OUT CONSTANT
	i_endoscopePose : ST_Frame;
	i_masterStatus :ST_MasterStatus;
	i_setupStatus: ST_SetupStatus;
	i_slaveArm :FB_SlaveArm;
END_VAR

VAR 
	jntIdx:INT;
	SDOSubIndexCur :WORD;
	armIdx:INT;
END_VAR
IF m_timePeriod > 1.0 THEN
	m_isFinished := TRUE;
END_IF

// reset instrument control box motor current limit
armIdx :=i_slaveArm.armIdx;
FOR jntIdx :=4 TO 8 DO
	//动力盒移动关节和器械旋转关节，共享一个控制字，由SDO写入
	IF (jntIdx=8)  THEN
		SDOSubIndexCur:=16#6098;
	//动力盒3、5号电机为一个驱动器，共享一个控制字，由SDO写入
	ELSIF (jntIdx=4) OR (jntIdx=6)  THEN
		SDOSubIndexCur:=16#6099;
	//动力盒2、4号电机为一个驱动器，共享一个控制字，由SDO写入
	ELSIF (jntIdx=5) OR (jntIdx=7)  THEN
		SDOSubIndexCur:=16#609A;
	END_IF

	// write max motor current if it changes and works in position mode  GVL_SlaveMotorParameters.g_motorMaxCurrent[jntIdx]
	m_MotorCurrentSDOWrite[jntIdx-3](sNetID:= GVL_SlaveJointEncoderCaliData.g_slaveArmNetID[armIdx],
					nSlaveAddr := GVL_SlaveJointEncoderCaliData.g_slaveJointNetPort[armIdx,jntIdx],
					nSubIndex:=0,nIndex:=SDOSubIndexCur,pSrcBuf:=ADR(m_wristJntRatedCurrent),
					cbBufLen:=SIZEOF(m_wristJntRatedCurrent),bExecute:=TRUE);
	IF NOT m_MotorCurrentSDOWrite[jntIdx-3].bBusy THEN
		m_MotorCurrentSDOWrite[jntIdx-3](bExecute:=FALSE);
	END_IF
	
END_FOR
END_METHOD

METHOD PUBLIC init : BOOL
VAR_IN_OUT CONSTANT
	i_slaveArm	:FB_SlaveArm;
END_VAR
VAR_IN_OUT 
	r_slaveArmCtrlCmd :ST_SlaveArmCtrlCmds;
END_VAR

VAR
	i:INT;
END_VAR
SUPER^.Init(i_slaveArm,r_slaveArmCtrlCmd);
m_jntEnableFlag:=g_zeroVec8i;

// update commands to arm
copyCmds(r_slaveArmCtrlCmd);
END_METHOD

END_FUNCTION_BLOCK

// ---- Mains/SlaveArmControl.TcPOU
PROGRAM SlaveArmControl
VAR
	
	// all data from other tasks and controller 
	m_nullSlaveInputDataPool : ST_SlaveInputDataPool;
	
	// flag to init robot
	m_robotInit :BOOL :=FALSE;
	
	// wait time before robot init  for ethercat to be statble 
	m_robotInitWaitTime : LREAL:=0;
	
	// slave robot
	m_slaveRobot:FB_SlaveRobot;

	// code execute time measure
	m_codeTime : Profiler;
	m_initMotorPID:FB_initMotorPID;
	m_initMotorPIDisFinished:BOOL;
END_VAR

m_codeTime(START:=TRUE, RESET:=TRUE);

// wait communication to be stable
IF(m_robotInitWaitTime<g_robotInitWaitTime) THEN
	m_robotInitWaitTime := m_robotInitWaitTime+g_slaveArmCtrlCycleTime;
	RETURN;
END_IF
//init motor pid
m_initMotorPIDisFinished:=m_initMotorPID.robotMotorRun();
IF NOT m_initMotorPIDisFinished THEN
	RETURN;
END_IF
// robot init
IF m_robotInit =FALSE OR GVL_InstruTestUIVars.g_powerBoxCalibrationFlag=FALSE THEN
	m_slaveRobot.Init();
	m_robotInit:=TRUE;
	GVL_InstruTestUIVars.g_powerBoxCalibrationFlag:=TRUE;
END_IF

// robot run
m_slaveRobot.run(m_nullSlaveInputDataPool);

//update UI data
UIProcessData();

m_codeTime(START:=FALSE);

METHOD UIProcessData : BOOL
VAR_INPUT
END_VAR
//update instrument chinese name 
GVL_InstruTestUIVars.g_instruNameCN := m_slaveRobot.m_slaveArms[1].instrument.instruTypeInfo.m_instruNameCH;
END_METHOD

END_PROGRAM

// ---- Sandbox/FB_SlaveCtrlInstruAutoTest_bak.TcPOU
// Brief: Slave Arm test
FUNCTION_BLOCK PUBLIC FB_SlaveCtrlInstruAutoTest_bak EXTENDS FB_SlaveArmCtrlBase
VAR CONSTANT
	m_instruOpenGripMoveTrajNum :INT :=18;
	m_instruGripMoveTrajNum :INT :=8;
	m_instruYawRange :LREAL := 75 * g_deg2Rad;
END_VAR
VAR
	// test mode. 
	//0: auto test - finger grip and release
	//1: auto test - finger open and mvoe
	//2: auto test - finger grip and move
	m_instruTestMode :INT := 0;
	m_lastInstruTestMode :INT := 0;
	
	// variables for auto test
	m_autoTestCycles :INT :=0;
	m_autoTestStep :INT :=0;

	// final target DH joint position and grip angle
	m_targetDHJntPos:Vec3d;
	m_targetGripAng:LREAL;
	m_targetGripForceLevel :LREAL :=0;
	
	// interploated command joint position and grip angle 
	m_cmdDHJntPos :Vec6d;
	m_cmdDHJntVel :Vec6d;
	m_cmdGripAng:LREAL;

	// last joint position 
	m_lastCmdJntPos :Vec8d ;
	
	// instrument controller
	m_instruController : FB_BasicInstruControl;
	m_usKnifeController : FB_UltrosonicKnifeControl;
	m_instruCmdJntPos,m_instruCmdJntVel : Vec5d;
	m_instruCmdJntTrq :Vec5d;
	
	// OTG
	m_DHJntOTG:ARRAY[1..3] OF FB_secOrdTrajFilter;
	m_gripAngleOTG : FB_secOrdTrajFilter;
	m_maxJntVel:Vec3d:=[3(2.0)];
	m_maxJntAcc:Vec3d:=[3(4.0)];
	
	// instrument open and grip move motion via points[roll, pitch, yaw]
	m_openGripStep :INT :=0;
	m_gripOpenStep :INT :=0;
	m_instruOpenGrioMovePos:ARRAY [1..m_instruOpenGripMoveTrajNum, 1..3] OF LREAL:=
	// move with gripper close
	[0,		-pi/2,		0,	
	0,		-pi/2,		pi/3,	
	0,		-pi/2,		-pi/3,
	0,		-pi/2+m_instruYawRange,		0,
	0,		-pi/2+m_instruYawRange,		pi/3,
	0,		-pi/2+m_instruYawRange,		-pi/3,
	0,		-pi/2-m_instruYawRange,		0,
	0,		-pi/2-m_instruYawRange,		-pi/3,
	0,		-pi/2-m_instruYawRange,		pi/3,
	// move with gripper open
	pi,		-pi/2,		0,	
	pi,		-pi/2,		pi/3,	
	pi,		-pi/2,		-pi/3,
	pi,		-pi/2+m_instruYawRange,		0,
	pi,		-pi/2+m_instruYawRange,		pi/3,
	pi,		-pi/2+m_instruYawRange,		-pi/3,
	pi,		-pi/2-m_instruYawRange,		0,
	pi,		-pi/2-m_instruYawRange,		-pi/3,
	pi,		-pi/2-m_instruYawRange,		pi/3];
	
	// instrument move motion via points[roll, pitch, yaw]
	m_instruGripMovePos:ARRAY [1..m_instruGripMoveTrajNum, 1..3] OF LREAL:=
	// move with gripper close
	[0,		-pi/2+m_instruYawRange,		pi/3,
	0,		-pi/2+m_instruYawRange,		-pi/3,
	0,		-pi/2-m_instruYawRange,		pi/3,
	0,		-pi/2-m_instruYawRange,		-pi/3,
	pi,		-pi/2+m_instruYawRange,		pi/3,
	pi,		-pi/2+m_instruYawRange,		-pi/3,
	pi,		-pi/2-m_instruYawRange,		pi/3,
	pi,		-pi/2-m_instruYawRange,		-pi/3];
	
	// instrument tyep
	m_instruType : E_InstrumentType;
																				
END_VAR

METHOD PROTECTED calcCmdJntPos : BOOL
VAR_IN_OUT CONSTANT
	i_endoscopePose : ST_Frame;
	i_masterStatus :ST_MasterStatus;
	i_setupStatus: ST_SetupStatus;
	i_slaveArm :FB_SlaveArm;
END_VAR

VAR 
	i:INT :=0;
	errThres :LREAL;

END_VAR

IF GVL_InstruTestUIVars.g_maxInstruAutoTestCycles > 0 AND m_autoTestCycles > GVL_InstruTestUIVars.g_maxInstruAutoTestCycles THEN
	RETURN;
END_IF

// determine final target DH joint position
CASE m_instruTestMode OF
	0:
		fingerOpenCloseTest(i_slaveArm);
	1:
		fingerOpenGripMoveTest(i_slaveArm);
	2:
		fingerGripMoveTest(i_slaveArm);
	ELSE
		RETURN;
END_CASE

// run OTG
FOR i:=1 TO 3  DO
	m_DHJntOTG[i].run(m_targetDHJntPos[i],0.0, o_cmdAcc=>,o_cmdVel=>m_cmdDHJntVel[i],o_cmdPos=> m_cmdDHJntPos[i+3]);
END_FOR
m_gripAngleOTG.run(m_targetGripAng,0.0, o_cmdAcc=>,o_cmdVel=>,o_cmdPos=>m_cmdGripAng);

// calculate target motor joint position from DH joint position
i_slaveArm.instrument.instruIK(m_cmdDHJntPos,m_cmdGripAng, o_jntPos=>m_cmdJntPos);

// command velocity
vecSub(m_cmdJntPos, m_lastCmdJntPos, m_cmdJntVel);
vecSelfMultiNum(m_cmdJntVel, g_slaveArmCtrlFreq);
m_lastCmdJntPos:=m_cmdJntPos;

m_lastInstruTestMode := m_instruTestMode;
END_METHOD

// override this function in each exact controller
METHOD PROTECTED calcCmdJntTrq : BOOL
VAR_IN_OUT CONSTANT
	i_endoscopePose : ST_Frame;
	i_masterStatus :ST_MasterStatus;
	i_setupStatus: ST_SetupStatus;
	i_slaveArm :FB_SlaveArm;
END_VAR

VAR 
	nullspaceMat :Mat7d;
	ctrlTrq : Vec7d;
	i : int ;
END_VAR
// set joint torque to zero in default
m_cmdJntTrq := g_zeroVec8d;

// instrument joint control
FOR i:=1 TO 5 DO 
	m_instruCmdJntPos[i]:=m_cmdJntPos[i+3];
	m_instruCmdJntVel[i]:=m_cmdJntVel[i+3];
END_FOR

IF i_slaveArm.instrument.instruType = InstruType_UltrasoundKnifeS OR i_slaveArm.instrument.instruType = InstruType_UltrasoundKnifeU THEN
	m_usKnifeController.run(m_instruCmdJntPos,m_instruCmdJntVel, m_targetGripForceLevel, i_slaveArm, o_cmdJntTrq=>m_instruCmdJntTrq);
ELSE
	m_instruController.run(m_instruCmdJntPos,m_instruCmdJntVel, m_cmdDHJntPos[6], m_cmdDHJntVel[6], m_targetGripForceLevel, i_slaveArm, o_cmdJntTrq=>m_instruCmdJntTrq);
END_IF

FOR i:=1 TO 5 DO
	m_cmdJntTrq[i+3]:=m_instruCmdJntTrq[i];
END_FOR
END_METHOD

METHOD fingerGripMoveTest : BOOL
VAR_IN_OUT CONSTANT
	i_slaveArm :FB_SlaveArm;
END_VAR
VAR
	i:INT;
END_VAR

m_targetGripForceLevel :=100;
m_autoTestStep := LIMIT(0,m_autoTestStep, m_instruGripMoveTrajNum-1);
FOR i:=1 TO 3 DO
	 m_targetDHJntPos[i] := m_instruGripMovePos[m_autoTestStep+1, i];
END_FOR
	 
IF ABS(m_cmdDHJntPos[4]-m_targetDHJntPos[1])< g_jntCtrlAngTolLow AND ABS(m_cmdDHJntPos[5]-m_targetDHJntPos[2])< g_jntCtrlAngTolLow 
		AND ABS(m_cmdDHJntPos[6]-m_targetDHJntPos[3])< g_jntCtrlAngTolLow  THEN
	m_autoTestStep :=m_autoTestStep + 1;
END_IF
 
IF m_autoTestStep >= m_instruGripMoveTrajNum THEN
	m_autoTestCycles := m_autoTestCycles + 1;
	m_autoTestStep := 0;
END_IF
END_METHOD

METHOD fingerGripOpenOnce : BOOL
VAR_IN_OUT CONSTANT
	i_slaveArm :FB_SlaveArm;
END_VAR
CASE m_gripOpenStep OF
	0:
		m_targetGripAng := 0;
		m_targetGripForceLevel :=0;
	1:
		m_targetGripAng := g_minSlaveGripAngle;
		m_targetGripForceLevel :=0;		
	2:
		m_targetGripAng := -45* g_deg2rad;
		m_targetGripForceLevel :=100;
	3:
		m_targetGripAng := g_minSlaveGripAngle;
		m_targetGripForceLevel :=100;

	4:
		m_targetGripAng := g_minSlaveGripAngle;
		m_targetGripForceLevel :=0;
END_CASE

IF ABS(m_cmdGripAng- m_targetGripAng)< g_jntCtrlAngTolLow THEN
	 m_gripOpenStep :=m_gripOpenStep + 1;
END_IF

fingerGripOpenOnce := m_gripOpenStep > 4;
END_METHOD

METHOD fingerOpenCloseTest : BOOL
VAR_IN_OUT CONSTANT
	i_slaveArm :FB_SlaveArm;
END_VAR
m_autoTestStep := LIMIT(0,m_autoTestStep, 5);
CASE m_autoTestStep OF
	0:
		m_targetGripAng := 0;
		m_targetGripForceLevel :=0;
	1:
		m_targetGripAng := GVL_InstruTestUIVars.g_maxGripAng * g_deg2Rad;//i_slaveArm.instrument.instruTypeInfo.m_maxGripAngle;
		m_targetGripForceLevel :=0;
	2:
		m_targetGripAng := g_minSlaveGripAngle;
		m_targetGripForceLevel :=0;
	3:
		m_targetGripAng := -pi/2;
		m_targetGripForceLevel :=100;
	4:
		m_targetGripAng := g_minSlaveGripAngle;
		m_targetGripForceLevel :=100;
	5:
		m_targetGripAng := 0;
		m_targetGripForceLevel :=0;
END_CASE

IF ABS(m_cmdGripAng- m_targetGripAng)< g_jntCtrlAngTolLow THEN
	 m_autoTestStep :=m_autoTestStep + 1;
END_IF

IF m_autoTestStep > 5 THEN
	m_autoTestCycles := m_autoTestCycles + 1;
	m_autoTestStep := 0;
END_IF
END_METHOD

METHOD fingerOpenGripMoveTest : BOOL
VAR_IN_OUT CONSTANT
	i_slaveArm :FB_SlaveArm;
END_VAR
VAR
	i:INT;
	fingerMotionFlag : BOOL;
END_VAR
m_autoTestStep := LIMIT(0,m_autoTestStep, m_instruOpenGripMoveTrajNum-1);
FOR i:=1 TO 3 DO
	 m_targetDHJntPos[i] := m_instruOpenGrioMovePos[m_autoTestStep+1, i];
END_FOR
	 
IF ABS(m_cmdDHJntPos[4]-m_targetDHJntPos[1])< g_jntCtrlAngTolLow AND ABS(m_cmdDHJntPos[5]-m_targetDHJntPos[2])< g_jntCtrlAngTolLow 
		AND ABS(m_cmdDHJntPos[6]-m_targetDHJntPos[3])< g_jntCtrlAngTolLow  THEN
	
	IF m_autoTestStep < m_instruOpenGripMoveTrajNum/2 THEN
		fingerMotionFlag:=fingerOpenGripOnce(i_slaveArm);
	ELSE
		fingerMotionFlag:=fingerGripOpenOnce(i_slaveArm);
	END_IF
	
	IF fingerMotionFlag THEN
		m_autoTestStep :=m_autoTestStep + 1;
		m_openGripStep :=0;
		m_gripOpenStep :=0;
	END_IF
	
END_IF
 
IF m_autoTestStep >= m_instruOpenGripMoveTrajNum THEN
	m_autoTestCycles := m_autoTestCycles + 1;
	m_autoTestStep := 0;
END_IF
END_METHOD

METHOD fingerOpenGripOnce : BOOL
VAR_IN_OUT CONSTANT
	i_slaveArm :FB_SlaveArm;
END_VAR
CASE m_openGripStep OF
	0:
		m_targetGripAng := 0;
		m_targetGripForceLevel :=0;
	1:
		m_targetGripAng := GVL_InstruTestUIVars.g_maxGripAng * g_deg2Rad;//i_slaveArm.instrument.instruTypeInfo.m_maxGripAngle;
		m_targetGripForceLevel :=0;
	2:
		m_targetGripAng := g_minSlaveGripAngle;
		m_targetGripForceLevel :=0;
	3:
		m_targetGripAng := -45 * g_deg2rad;
		m_targetGripForceLevel :=100;
	4:
		m_targetGripAng := g_minSlaveGripAngle;
		m_targetGripForceLevel :=100;
END_CASE

IF ABS(m_cmdGripAng- m_targetGripAng)< g_jntCtrlAngTolLow THEN
	 m_openGripStep :=m_openGripStep + 1;
END_IF

fingerOpenGripOnce := m_openGripStep > 4;
END_METHOD

METHOD PUBLIC init : BOOL
VAR_IN_OUT CONSTANT
	i_slaveArm	:FB_SlaveArm;
END_VAR
VAR_IN_OUT 
	r_slaveArmCtrlCmd :ST_SlaveArmCtrlCmds;
END_VAR

VAR
	i:int;
END_VAR
SUPER^.Init(i_slaveArm,r_slaveArmCtrlCmd);
m_lastCmdJntPos:=m_cmdJntPos;
m_jntOPMode[1] := DriverOPMode_PosTrq;
m_jntOPMode[2] := DriverOPMode_PosTrq;
m_jntOPMode[3] := DriverOPMode_PosTrq;
m_jntOPMode[4] := DriverOPMode_Trq;
m_jntOPMode[5] := DriverOPMode_Trq;
m_jntOPMode[6] := DriverOPMode_Trq;
m_jntOPMode[7] := DriverOPMode_Trq;
m_jntOPMode[8] := DriverOPMode_Trq;

m_instruTestMode := GVL_InstruTestUIVars.g_instruAutoTestMode;
m_autoTestStep:=0 ;
m_autoTestCycles := 0;
m_openGripStep :=0;
m_gripOpenStep :=0;
m_cmdDHJntPos :=i_slaveArm.curDHJntPos;
m_cmdDHJntVel :=g_zeroVec6d;
m_targetGripAng := i_slaveArm.curGripAngle;
m_targetDHJntPos[1] := i_slaveArm.curDHJntPos[4];
m_targetDHJntPos[2] := i_slaveArm.curDHJntPos[5];
m_targetDHJntPos[3] := i_slaveArm.curDHJntPos[6];

// init instrument controller
m_instruController.init(i_slaveArm);
m_usKnifeController.init(i_slaveArm);
m_instruType := i_slaveArm.instrument.instruType;

FOR i:=1 TO 3  DO
	m_DHJntOTG[i].init(m_cmdDHJntPos[i+3], 0, m_maxJntVel[i], m_maxJntAcc[i], g_slaveArmCtrlCycleTime);
END_FOR

m_gripAngleOTG.init(m_targetGripAng, 0, m_maxJntVel[3], m_maxJntAcc[3], g_slaveArmCtrlCycleTime);
// update commands to arm
copyCmds(r_slaveArmCtrlCmd);
END_METHOD

PROPERTY InstruBacklash : Vec5d
GET
IF m_instruType = InstruType_UltrasoundKnifeS OR m_instruType = InstruType_UltrasoundKnifeU THEN
	instruBacklash := g_zeroVec5d;
ELSE
	instruBacklash := m_instruController.m_jntBacklash;
END_IF
END_GET
END_PROPERTY

END_FUNCTION_BLOCK

// ---- Sandbox/FB_SlaveCtrlInstruVerify_bak.TcPOU
// Brief: Slave Arm test
FUNCTION_BLOCK PUBLIC FB_SlaveCtrlInstruVerify_bak EXTENDS FB_SlaveArmCtrlBase
VAR CONSTANT
	m_instruVerifyTrajNum :INT :=12;
END_VAR
VAR
	// rising edge generator for instrument information reading
	m_nextStepRTrig:R_TRIG;
	m_lastStepRTrig:R_TRIG;
											
	// variable for instument veify
	m_verifyTestStep :INT :=0;
	m_reachVerifyPos : BOOL := FALSE;
	// instrument move motion via points[roll, pitch, yaw]
	m_instruVerifyPos:ARRAY [1..m_instruVerifyTrajNum, 1..4] OF LREAL:= 
	[	0,  -pi/2 + pi/3,	0,	0,
		0,  -pi/2 - pi/3,	0,	0,
		0,  -pi/2,	0,	0,
		0,  -pi/2 ,	pi/3,	0,
		0,  -pi/2,	-pi/3,	0,
		pi,  -pi/2 ,	0,	0,
		0,  -pi/2 ,	0,	0,
		0,  -pi/2 ,	0,	pi,
		0,  -pi/2 ,	0,	0,
		0,  -pi/2 ,	0,	-pi/3,
		0,	-pi/2,	0, 	0];
				

	// final target DH joint position and grip angle
	m_targetDHJntPos:Vec3d;
	m_targetGripAng:LREAL;
	m_targetGripForceLevel :LREAL :=0;
	
	// interploated command joint position and grip angle 
	m_cmdDHJntPos :Vec6d;
	m_cmdDHJntVel :Vec6d;
	m_cmdGripAng:LREAL;

	// last joint position 
	m_lastCmdJntPos :Vec8d ;
	
	// instrument controller
	m_instruController : FB_BasicInstruControl;
	m_usKnifeController : FB_UltrosonicKnifeControl;
	m_instruCmdJntPos,m_instruCmdJntVel : Vec5d;
	m_instruCmdJntTrq :Vec5d;
	
	// OTG
	m_DHJntOTG:ARRAY[1..3] OF FB_secOrdTrajFilter;
	m_gripAngleOTG : FB_secOrdTrajFilter;
	m_maxJntVel:Vec3d:=[3(2.0)];
	m_maxJntAcc:Vec3d:=[3(4.0)];
	
	// instrument tyep
	m_instruType : E_InstrumentType;

END_VAR

METHOD PROTECTED calcCmdJntPos : BOOL
VAR_IN_OUT CONSTANT
	i_endoscopePose : ST_Frame;
	i_masterStatus :ST_MasterStatus;
	i_setupStatus: ST_SetupStatus;
	i_slaveArm :FB_SlaveArm;
END_VAR

VAR 
	i:INT :=0;
	errThres :LREAL;

END_VAR
// determine final target DH joint position
instruVerifyTest(i_slaveArm);

// run OTG
FOR i:=1 TO 3  DO
	m_DHJntOTG[i].run(m_targetDHJntPos[i],0.0, o_cmdAcc=>,o_cmdVel=>m_cmdDHJntVel[i],o_cmdPos=> m_cmdDHJntPos[i+3]);
END_FOR
m_gripAngleOTG.run(m_targetGripAng,0.0, o_cmdAcc=>,o_cmdVel=>,o_cmdPos=>m_cmdGripAng);

// calculate target motor joint position from DH joint position
i_slaveArm.instrument.instruIK(m_cmdDHJntPos,m_cmdGripAng, o_jntPos=>m_cmdJntPos);

// command velocity
vecSub(m_cmdJntPos, m_lastCmdJntPos, m_cmdJntVel);
vecSelfMultiNum(m_cmdJntVel, g_slaveArmCtrlFreq);
m_lastCmdJntPos:=m_cmdJntPos;
END_METHOD

// override this function in each exact controller
METHOD PROTECTED calcCmdJntTrq : BOOL
VAR_IN_OUT CONSTANT
	i_endoscopePose : ST_Frame;
	i_masterStatus :ST_MasterStatus;
	i_setupStatus: ST_SetupStatus;
	i_slaveArm :FB_SlaveArm;
END_VAR

VAR 
	nullspaceMat :Mat7d;
	ctrlTrq : Vec7d;
	i : int ;
END_VAR
// set joint torque to zero in default
m_cmdJntTrq := g_zeroVec8d;

// instrument joint control
FOR i:=1 TO 5 DO 
	m_instruCmdJntPos[i]:=m_cmdJntPos[i+3];
	m_instruCmdJntVel[i]:=m_cmdJntVel[i+3];
END_FOR

IF i_slaveArm.instrument.instruType = InstruType_UltrasoundKnifeS OR i_slaveArm.instrument.instruType = InstruType_UltrasoundKnifeU THEN
	m_usKnifeController.run(m_instruCmdJntPos,m_instruCmdJntVel, m_targetGripForceLevel, i_slaveArm, o_cmdJntTrq=>m_instruCmdJntTrq);
ELSE
	m_instruController.run(m_instruCmdJntPos,m_instruCmdJntVel, m_cmdDHJntPos[6], m_cmdDHJntVel[6], m_targetGripForceLevel, i_slaveArm, o_cmdJntTrq=>m_instruCmdJntTrq);
END_IF

FOR i:=1 TO 5 DO
	m_cmdJntTrq[i+3]:=m_instruCmdJntTrq[i];
END_FOR
END_METHOD

METHOD PUBLIC init : BOOL
VAR_IN_OUT CONSTANT
	i_slaveArm	:FB_SlaveArm;
END_VAR
VAR_IN_OUT 
	r_slaveArmCtrlCmd :ST_SlaveArmCtrlCmds;
END_VAR

VAR
	i:int;
END_VAR
SUPER^.Init(i_slaveArm,r_slaveArmCtrlCmd);
m_lastCmdJntPos:=m_cmdJntPos;
m_jntOPMode[1] := DriverOPMode_PosTrq;
m_jntOPMode[2] := DriverOPMode_PosTrq;
m_jntOPMode[3] := DriverOPMode_PosTrq;
m_jntOPMode[4] := DriverOPMode_Trq;
m_jntOPMode[5] := DriverOPMode_Trq;
m_jntOPMode[6] := DriverOPMode_Trq;
m_jntOPMode[7] := DriverOPMode_Trq;
m_jntOPMode[8] := DriverOPMode_Trq;

m_verifyTestStep := 0;
m_cmdDHJntPos :=i_slaveArm.curDHJntPos;
m_cmdDHJntVel :=g_zeroVec6d;
m_targetGripAng := i_slaveArm.curGripAngle;
m_targetDHJntPos[1] := i_slaveArm.curDHJntPos[4];
m_targetDHJntPos[2] := i_slaveArm.curDHJntPos[5];
m_targetDHJntPos[3] := i_slaveArm.curDHJntPos[6];

// init instrument controller
m_instruController.init(i_slaveArm);
m_usKnifeController.init(i_slaveArm);

FOR i:=1 TO 3  DO
	m_DHJntOTG[i].init(m_cmdDHJntPos[i+3], 0, m_maxJntVel[i], m_maxJntAcc[i], g_slaveArmCtrlCycleTime);
END_FOR

m_gripAngleOTG.init(m_targetGripAng, 0, 2*m_maxJntVel[3], 2*m_maxJntAcc[3], g_slaveArmCtrlCycleTime);
// update commands to arm
copyCmds(r_slaveArmCtrlCmd);
END_METHOD

PROPERTY InstruBacklash : Vec5d
GET
IF m_instruType = InstruType_UltrasoundKnifeS OR m_instruType = InstruType_UltrasoundKnifeU THEN
	instruBacklash := g_zeroVec5d;
ELSE
	instruBacklash := m_instruController.m_jntBacklash;
END_IF
END_GET
END_PROPERTY

METHOD instruVerifyTest : BOOL
VAR_IN_OUT CONSTANT
	i_slaveArm :FB_SlaveArm;
END_VAR
VAR
	i:INT;
	nextStepFlag :BOOL;
	lastStepFlag :BOOL;
END_VAR
m_targetGripForceLevel :=0;
m_verifyTestStep := LIMIT(0,m_verifyTestStep, m_instruVerifyTrajNum-1);

FOR i:=1 TO 3 DO
	 m_targetDHJntPos[i] := m_instruVerifyPos[m_verifyTestStep+1, i];
END_FOR
 m_targetGripAng := LIMIT(0, m_instruVerifyPos[m_verifyTestStep+1,4], i_slaveArm.instrument.instruTypeInfo.m_maxGripAngle);

m_nextStepRTrig(CLK:= GVL_InstruTestUIVars.g_instruVerifyNextStepFlag, Q=>nextStepFlag );
m_lastStepRTrig(CLK:= GVL_InstruTestUIVars.g_instruVerifyLastStepFlag, Q=>lastStepFlag );
IF  nextStepFlag THEN
	m_verifyTestStep :=m_verifyTestStep + 1;
ELSIF  lastStepFlag THEN
	m_verifyTestStep :=m_verifyTestStep - 1;
END_IF
END_METHOD

END_FUNCTION_BLOCK

// ---- Sandbox/FB_SlaveCtrlMasterSlave_backup.TcPOU
// Brief: Slave Arm MasterSlave controller
FUNCTION_BLOCK PUBLIC FB_SlaveCtrlMasterSlave_backup EXTENDS FB_SlaveArmCtrlBase
VAR_INPUT
END_VAR
VAR_OUTPUT
END_VAR
VAR
	// minimum distance between instrument tip and remote center
	m_minInstruRCDis:LREAL := 0.05;
	
	// master-slave motion scale
	m_MSMotionScale :LREAL;
		
	// gripper match angle threshold
	m_gripperMatchAngThres :LREAL := 2*g_deg2Rad;
	
	// control error thershold from joint limit back to free space
	m_maxPosTrackErr :LREAL := 0.05;
	m_maxOriTrackErr :LREAL :=g_deg2Rad * 5;
	
	// filter cut-off frequency for master-slave control
	m_macroCmdJntPosLpfCutoffFreq : LREAL :=5;
	m_microCmdJntPosLpfCutoffFreq : LREAL :=15;
	
	// last command joint position
	m_lastCmdJntPos :Vec8d;
	
	// simulated DH joint position
	m_simDHJntPos : Vec6d;
	
	// simulated slave twist of DH joint
	m_simDHJointVel :Vec6d;
		
	// enter master-slave control for the first time
	m_firstIn :BOOL := TRUE;
	
	// flag if reach joint limit
	m_reachMacroJntLimit :BOOL;
	m_reachWristJntLimit :BOOL;
	
	// master/slave origin pose when first enter master-slave control
	m_masterOriginPose : ST_Frame;
	m_slaveOriginPose : ST_Frame;
	
	// orientation deviation(in master coordinate) between master and slave when first enter control
	m_MSOriDeviation : Mat3d;
	
	// command joint position filter
	m_cmdJntPosLpf:ARRAY[1..8] OF FB_LowPassFilter;
	
	// commmand yaw angle and velocity
	m_cmdYawAngle :LREAL;
	m_cmdYawVel :LREAL;
	
	// comand yaw angle and velocity filter
	m_cmdYawAngLpf : FB_LowPassFilter;
	m_cmdYawVelLpf : FB_LowPassFilter;
	
	// master pose/velocity in monitor coordinate
	m_masterPose :ST_Frame;
	m_masterTwist : Vec6d;
	
	// master grip angle
	m_masterGripAngle : LREAL;
	
	// slave command/current pose in endoscope coordinate
	m_slaveCmdPoseInScope :ST_Frame;
	m_slavePoseInScope : ST_Frame;
	
	// slave command/current pose in cart
	m_slaveCmdPoseInCart :ST_Frame;
	m_slavePoseInCart : ST_Frame;
	
	// instrument controller
	m_basicInstruController : FB_BasicInstruControl;
	m_usKnifeController : FB_UltrosonicKnifeControl;
	
	// slave command grip angle and grip force level
	m_slaveCmdGripAngle :LREAL;
	m_slaveCmdGripForceLevel:LREAL;
	
	// slave pose error
	m_slavePosErr :Vec3d;
	m_slaveRotErr :Mat3d;
	m_errAngle : LREAL;
	m_errAxisLocal, m_errAxis :Vec3d;
	m_masterSlavePoseError :Vec6d;
	
	// velocity for slave to track master motion
	m_slaveTrackTwist :Vec6d;
	m_slaveCmdVel, m_slaveCmdWVel : Vec3d;
	
	// last master gripper angle
	m_lastMasterGripAngle :LREAL;
	
	// master gripper angle velocity
	m_masterGripAngleVel :LREAL;
	m_masterGripAngleVelLpf :FB_LowPassFilter;
	
	// flag to start gripper control
	m_gripperCtrlFlag :BOOL;
	
	// code execute time measure
	m_codeTime : Profiler;
	
END_VAR

METHOD PROTECTED calcCmdJntPos : BOOL
VAR_IN_OUT CONSTANT
	i_endoscopePose : ST_Frame;
	i_masterStatus :ST_MasterStatus;
	i_setupStatus: ST_SetupStatus;
	i_slaveArm :FB_SlaveArm;
END_VAR

VAR 
	i,j : INT;
	tmpMat3d : Mat3d;
	masterMotionRange : Vec3d;
	
	masterVelInScope, masterWVelInScope :Vec3d;
	masterVelInCart, masterWVelInCart :Vec3d;

	cmdVelScale :LREAL;
	invJaco :Mat6d;
	DHJntCmdDeltaPos :Vec6d;
	armJntJaco,armJntJacoInv, wristJntJaco :Mat3d;
	velByWristJnt,velByArmJnt : Vec3d;
	armDHJntVel, wristDHJntVel :Vec3d;
	tmpFrame : ST_Frame;
	slaveSimDHJntPos :Vec6d;
	jnt3Limit :LREAL;
END_VAR
m_codeTime(START:=TRUE, RESET:=TRUE);

IF isFinished THEN
	RETURN;
END_IF

// decide matched master arm index
FOR i:=1 TO g_mArmNum DO 
	IF i_masterStatus.m_teleSlaveArmIdx[i] = i_slaveArm.armIdx THEN
		m_masterPose := i_masterStatus.m_curArmPose[i];
		m_masterTwist := i_masterStatus.m_curArmTwist[i];
		m_masterGripAngle := i_masterStatus.m_gripAngle[i];
	END_IF
END_FOR

// compute slave pose in endoscope coordinate
m_slavePoseInCart := transform(i_setupStatus.m_curEndPose[i_slaveArm.armIdx], i_slaveArm.simCartPose);
tmpFrame :=invFrame(i_endoscopePose);
m_slavePoseInScope := transform(tmpFrame, m_slavePoseInCart);

// handle for the first time in
IF TRUE = m_firstIn THEN
	m_firstIn := FALSE;
	m_masterOriginPose :=m_masterPose;
	m_slaveOriginPose := m_slavePoseInScope;
	matTranspose(m_masterOriginPose.m_rot, tmpMat3d);
	matMultiply(tmpMat3d, m_slavePoseInScope.m_rot,m_MSOriDeviation);
	m_lastMasterGripAngle := m_masterGripAngle;
	
	// only update motion scale while entering teleControl 
	m_MSMotionScale := 1.0/ MAX(1,  i_masterStatus.m_motionScale);
END_IF

// compute master twist in slave arm coordinate
(*FOR i:=1 TO 3 DO
	masterVelInScope[i] := m_masterTwist[i]*i_masterStatus.m_motionScale;
	masterWVelInScope[i] := m_masterTwist[i+3];
END_FOR
matMultiVec(i_endoScopePose.m_rot, masterVelInScope, masterVelInCart);
matMultiVec(i_endoScopePose.m_rot, masterWVelInScope, masterWVelInCart);
matTranspose(i_setupStatus.m_curEndPose[i_slaveArm.armIdx].m_rot, tmpMat3d);
matMultiVec(tmpMat3d,masterVelInCart, m_masterFFVel);
matMultiVec(tmpMat3d,masterWVelInCart, m_masterFFWVel);
FOR i:=1 TO 3 DO
	m_cmdCartTwist[i] := m_masterFFVel[i];
	m_cmdCartTwist[i+3] := m_masterFFWVel[i];
END_FOR*)

// compute slave command pose in scope
vecSub(m_masterPose.m_pos, m_masterOriginPose.m_pos, masterMotionRange);

vecSelfMultiNum(masterMotionRange, m_MSMotionScale);
vecAdd(m_slaveOriginPose.m_pos, masterMotionRange, m_slaveCmdPoseInScope.m_pos);
matMultiply(m_masterPose.m_rot, m_MSOriDeviation, m_slaveCmdPoseInScope.m_rot);

// compute slave command pose in slave arm coordinate
m_slaveCmdPoseInCart := transform(i_endoScopePose, m_slaveCmdPoseInScope);
tmpFrame := invFrame(i_setupStatus.m_curEndPose[i_slaveArm.armIdx]);
m_cmdCartPose := transform(tmpFrame, m_slaveCmdPoseInCart);

// compute pose error
vecSub(m_cmdCartPose.m_pos, i_slaveArm.simCartPose.m_pos, m_slavePosErr);

matTranspose(i_slaveArm.simCartPose.m_rot, tmpMat3d);
matMultiply(tmpMat3d, m_cmdCartPose.m_rot, m_slaveRotErr);
rot2AngAxis(m_slaveRotErr, angle=>m_errAngle, axis=>m_errAxisLocal);
matMultiVec(i_slaveArm.simCartPose.m_rot, m_errAxisLocal, m_errAxis);

// calculate pose error in endoscope
calcMSErrInScope(i_endoscopePose, i_setupStatus.m_curEndPose[i_slaveArm.armIdx], i_slaveArm);

// safety check
(*IF norm(m_slavePosErr) > m_maxPosTrackErr OR ABS(m_errAngle)>m_maxOriTrackErr THEN
	m_isFinished := TRUE;
END_IF*) 

// pose track control
vecMultiNum(m_slavePosErr, g_slaveArmCtrlFreq, m_slaveCmdVel);
vecMultiNum(m_errAxis, m_errAngle*g_slaveArmCtrlFreq, m_slaveCmdWVel);
FOR i:=1 TO 3 DO 
	m_slaveTrackTwist[i] := m_slaveCmdVel[i];
	m_slaveTrackTwist[i+3] := m_slaveCmdWVel[i];
END_FOR

// compute command velocity for DH joints
invJaco := i_slaveArm.simJacoInv;
matMultiVec(invJaco, m_slaveTrackTwist, m_simDHJointVel);

// limit DH joints velocity 
cmdVelScale := 1;
FOR i:=1 TO g_cartDofs DO 
	cmdVelScale:=MAX(cmdVelScale, ABS(m_simDHJointVel[i]/GVL_SlaveMotorParameters.g_maxJntVel[i]));
END_FOR
vecSelfMultiNum(m_simDHJointVel, 1.0/cmdVelScale);
vecSelfMultiNum(m_slaveTrackTwist, 1.0/cmdVelScale);
vecSelfMultiNum(m_slaveCmdVel, 1.0/cmdVelScale);
vecSelfMultiNum(m_slaveCmdWVel, 1.0/cmdVelScale);

FOR i:=1 TO 3 DO
	armDHJntVel[i]:=m_simDHJointVel[i];
	wristDHJntVel[i]:=m_simDHJointVel[i+3];
END_FOR

// limit instrument wrist dofs
limitInstruDofs(i_slaveArm, wristDHJntVel);

// limit instrument wrist joint position
IF  (m_reachWristJntLimit AND ABS(m_errAngle)>m_maxOriTrackErr) THEN
	wristDHJntVel:=g_zeroVec3d;
	m_reachWristJntLimit:=TRUE;
ELSE
	m_reachWristJntLimit :=FALSE;
	FOR i:=1 TO 3 DO
		IF (wristDHJntVel[i] > 0 AND i_slaveArm.simDHJntPos[i+3] + wristDHJntVel[i]*g_slaveArmCtrlCycleTime> i_slaveArm.instrument.instruTypeInfo.m_wristMaxDHJntPos[i]) OR 
			(wristDHJntVel[i]<0 AND i_slaveArm.simDHJntPos[i+3] + wristDHJntVel[i]*g_slaveArmCtrlCycleTime< i_slaveArm.instrument.instruTypeInfo.m_wristMinDHJntPos[i])  THEN
			wristDHJntVel:=g_zeroVec3d;
			m_reachWristJntLimit:=TRUE;
			CONTINUE;
		END_IF
	END_FOR
END_IF

// modify arm joints velocity to compensate wrist joint motion
FOR i:=1 TO 3 DO
	FOR j:=1 TO 3 DO
		armJntJaco[i,j]:=i_slaveArm.simJaco[i,j];
		wristJntJaco[i,j]:=i_slaveArm.simJaco[i,j+3];
	END_FOR
END_FOR
invMat3(armJntJaco, armJntJacoInv);
matMultiVec(wristJntJaco, wristDHJntVel, velByWristJnt);
vecSub(m_slaveCmdVel, velByWristJnt, velByArmJnt);
matMultiVec(armJntJacoInv, velByArmJnt, armDHJntVel);

// limit DH joints velocity 
cmdVelScale := 1;
FOR i:=1 TO 3 DO 
	cmdVelScale:=MAX(cmdVelScale, ABS(armDHJntVel[i]/GVL_SlaveMotorParameters.g_maxJntVel[i]));
END_FOR
vecSelfMultiNum(armDHJntVel, 1.0/cmdVelScale);

// limit arm joint position
m_reachMacroJntLimit :=FALSE;
FOR i:=1 TO 3 DO
	IF (armDHJntVel[i] > 0 AND  i_slaveArm.simDHJntPos[i] + armDHJntVel[i]*g_slaveArmCtrlCycleTime> GVL_SlaveMotorParameters.g_maxDHJntPos[i]) OR 
		(armDHJntVel[i] <0 and	i_slaveArm.simDHJntPos[i] + armDHJntVel[i]*g_slaveArmCtrlCycleTime< GVL_SlaveMotorParameters.g_minDHJntPos[i]) THEN
		armDHJntVel[i]:=0;
		m_reachMacroJntLimit:=TRUE;
	END_IF
END_FOR

// joint 3 up limit to remote center
jnt3Limit := i_slaveArm.instrument.instruTypeInfo.m_rodLength+i_slaveArm.instrument.instruTypeInfo.m_headLength
											+ i_slaveArm.instrument.instruTypeInfo.m_fingerLength - GVL_SlaveArmKinematic.g_minInstruRCDis;
IF (armDHJntVel[3] > 0 AND i_slaveArm.simDHJntPos[3] + armDHJntVel[3]*g_slaveArmCtrlCycleTime> jnt3Limit) THEN
	armDHJntVel[3]:=0;
	m_reachMacroJntLimit:=TRUE;
END_IF

// integrate command DH joint position
FOR i:=1 TO 3 DO
	m_simDHJointVel[i]:=armDHJntVel[i];
	m_simDHJointVel[i+3]:=wristDHJntVel[i];
END_FOR
vecMultiNum(m_simDHJointVel, g_slaveArmCtrlCycleTime, DHJntCmdDeltaPos);
slaveSimDHJntPos:=i_slaveArm.simDHJntPos;
vecAdd(slaveSimDHJntPos, DHJntCmdDeltaPos, m_simDHJntPos);

// gripper angle/force control
gripperControl(i_slaveArm);

// calculate target motor joint position/velocity from DH joint position
i_slaveArm.instrument.instruIK(m_simDHJntPos,m_slaveCmdGripAngle, o_jntPos=>m_simJntPos);

// filt command joint position
FOR i:=1 TO g_sJntNum DO 
	m_cmdJntPos[i] := m_cmdJntPosLpf[i].run(m_simJntPos[i]);
END_FOR

// compute command joint velocity
vecSub(m_cmdJntPos, m_lastCmdJntPos, m_cmdJntVel);
vecSelfMultiNum(m_cmdJntVel, g_slaveArmCtrlFreq);
m_lastCmdJntPos:=m_cmdJntPos;

m_codeTime(START:=FALSE);
END_METHOD

// override this function in each exact controller
METHOD PROTECTED calcCmdJntTrq : BOOL
VAR_IN_OUT CONSTANT
	i_endoscopePose : ST_Frame;
	i_masterStatus :ST_MasterStatus;
	i_setupStatus: ST_SetupStatus;
	i_slaveArm :FB_SlaveArm;
END_VAR
VAR
	i :INT ;
	instruCmdGripAngle, instruCmdGripForceLevel :LREAL;
	instruCmdJntPos, instruCmdJntVel : Vec5d;	
	instruJntCtrlTrq :Vec5d;
END_VAR
IF isFinished THEN
	RETURN;
END_IF

// set joint torque to zero in default
m_cmdJntTrq := g_zeroVec8d;

// instrument joint control
FOR i:=1 TO 5 DO 
	instruCmdJntPos[i]:=m_cmdJntPos[i+3];
	instruCmdJntVel[i]:=m_cmdJntVel[i+3];
END_FOR
m_cmdYawAngle := m_cmdYawAngLpf.run(m_simDHJntPos[6]);
m_cmdYawVel := m_cmdYawVelLpf.run(m_simDHJointVel[6]);

IF i_slaveArm.instrument.instruType = InstruType_UltrasoundKnifeS OR i_slaveArm.instrument.instruType = InstruType_UltrasoundKnifeU THEN
	m_usKnifeController.run(instruCmdJntPos,instruCmdJntVel, m_slaveCmdGripForceLevel, i_slaveArm, o_cmdJntTrq=>instruJntCtrlTrq);
ELSE
	m_basicInstruController.run(instruCmdJntPos,instruCmdJntVel, m_cmdYawAngle, m_cmdYawVel, m_slaveCmdGripForceLevel, i_slaveArm, o_cmdJntTrq=>instruJntCtrlTrq);
END_IF

FOR i:=1 TO 5 DO
	m_cmdJntTrq[i+3]:=instruJntCtrlTrq[i];
END_FOR
END_METHOD

METHOD calcMSErrInScope : BOOL
VAR_IN_OUT CONSTANT
	i_endoscopePose : ST_Frame;
	i_setupPose :ST_Frame;
	i_slaveArm :FB_SlaveArm;
END_VAR
VAR
	posErrInCart,oriErrInCart :Vec3d;
	invRot :Mat3d;
	posErrInScope,oriErrInScope :Vec3d;
	i:INT;
END_VAR
m_masterSlavePoseError := g_zeroVec6d;

// pose error caused by joints limits
IF m_reachMacroJntLimit OR m_reachWristJntLimit THEN
	// pose error in cart coordinate
	matMultiVec(i_setupPose.m_rot, m_slavePosErr, posErrInCart);
	matMultiVec(i_setupPose.m_rot, m_errAxis, oriErrInCart);
	vecSelfMultiNum(oriErrInCart, m_errAngle);
	
	// pose err in endoscope coordinate
	matTranspose(i_endoscopePose.m_rot, invRot);
	matMultiVec(invRot, posErrInCart, posErrInScope);
	matMultiVec(invRot, oriErrInCart, oriErrInScope);
	
	FOR i:=1 TO 3 DO 
		m_masterSlavePoseError[i]:=posErrInScope[i];
	END_FOR
	
	FOR i:=1 TO 3 DO 
		m_masterSlavePoseError[i+3]:=oriErrInScope[i];
	END_FOR

END_IF
END_METHOD

METHOD gripperControl : BOOL
VAR_IN_OUT CONSTANT
	i_slaveArm :FB_SlaveArm;
END_VAR

VAR
	matchedSlaveGripAngle:LREAL;
	matchedSlaveGripForce:LREAL;
	masterGripVelThres :LREAL := 5.0 *g_deg2Rad;
END_VAR
// compute master grip veloicty
m_masterGripAngleVel:= (m_masterGripAngle - m_lastMasterGripAngle)/g_slaveArmCtrlCycleTime;
m_masterGripAngleVel := m_masterGripAngleVelLpf.run(m_masterGripAngleVel);
m_lastMasterGripAngle :=m_masterGripAngle;

// compute matched slave grip angle and force
i_slaveArm.instrument.gripAngleMap(m_masterGripAngle,o_instruGripAngle=>matchedSlaveGripAngle, o_instruGripForceLevel=>matchedSlaveGripForce);

IF m_gripperCtrlFlag THEN
	m_slaveCmdGripAngle := matchedSlaveGripAngle;
	m_slaveCmdGripForceLevel := matchedSlaveGripForce;
	RETURN;
ELSE
	//m_gripperCtrlFlag := (ABS(m_masterGripAngleVel) >masterGripVelThres) AND  (m_masterGripAngleVel * (matchedSlaveGripAngle-i_slaveArm.curGripAngle)>0);
	m_gripperCtrlFlag := ABS(matchedSlaveGripAngle-i_slaveArm.curGripAngle)<m_gripperMatchAngThres OR 
	     (matchedSlaveGripAngle>=i_SlaveArm.instrument.instruTypeInfo.m_maxGripAngle - m_gripperMatchAngThres AND i_slaveArm.curGripAngle>=matchedSlaveGripAngle) OR 
		(matchedSlaveGripAngle<=i_SlaveArm.instrument.instruTypeInfo.m_minGripAngle + m_gripperMatchAngThres AND i_slaveArm.curGripAngle<=matchedSlaveGripAngle);
END_IF
END_METHOD

METHOD PUBLIC init : BOOL
VAR_IN_OUT CONSTANT
	i_slaveArm	:FB_SlaveArm;
END_VAR
VAR_IN_OUT 
	r_slaveArmCtrlCmd :ST_SlaveArmCtrlCmds;
END_VAR
VAR 
	i :INT ;
END_VAR
SUPER^.Init(i_slaveArm,r_slaveArmCtrlCmd);
m_simJntPos :=m_cmdJntPos;
m_lastCmdJntPos :=m_cmdJntPos;
m_jntOPMode[1] := DriverOPMode_PosTrq;
m_jntOPMode[2] := DriverOPMode_PosTrq;
m_jntOPMode[3] := DriverOPMode_PosTrq;
m_jntOPMode[4] := DriverOPMode_Trq;
m_jntOPMode[5] := DriverOPMode_Trq;
m_jntOPMode[6] := DriverOPMode_Trq;
m_jntOPMode[7] := DriverOPMode_Trq;
m_jntOPMode[8] := DriverOPMode_Trq;
m_firstIn :=TRUE;
m_gripperCtrlFlag :=false;

// init gripper angle
m_slaveCmdGripAngle := i_slaveArm.curGripAngle;
m_slaveCmdGripForceLevel:=0;

// init filter
FOR i:=1 TO 3 DO
	m_cmdJntPosLpf[i].init(1, m_macroCmdJntPosLpfCutoffFreq, g_slaveArmCtrlFreq);
END_FOR
FOR i:=4 TO g_sJntNum DO
	m_cmdJntPosLpf[i].init(1, m_microCmdJntPosLpfCutoffFreq, g_slaveArmCtrlFreq);
END_FOR
m_cmdYawAngLpf.init(1, m_microCmdJntPosLpfCutoffFreq, g_slaveArmCtrlFreq);
m_cmdYawVelLpf.init(1, m_microCmdJntPosLpfCutoffFreq, g_slaveArmCtrlFreq);
m_masterGripAngleVelLpf.init(1, m_microCmdJntPosLpfCutoffFreq, g_slaveArmCtrlFreq);

// init controller
m_basicInstruController.init(i_slaveArm);
m_usKnifeController.init(i_slaveArm);

// update commands to arm
copyCmds(r_slaveArmCtrlCmd);
END_METHOD

// limit specific joint dofs based on instrument types
METHOD PRIVATE limitInstruDofs : BOOL
VAR_IN_OUT CONSTANT
	i_slaveArm :FB_SlaveArm;
END_VAR

VAR_IN_OUT
	r_wristDHJntVel :Vec3d;
END_VAR
IF i_slaveArm.instrument.instruType = InstruType_UltrasoundKnifeS OR i_slaveArm.instrument.instruType = InstruType_UltrasoundKnifeU THEN
	r_wristDHJntVel[2] :=0;
	r_wristDHJntVel[3] :=0;
END_IF
END_METHOD

PROPERTY masterSlavePoseErr : REFERENCE to Vec6d
GET
masterSlavePoseErr REF= m_masterSlavePoseError;
END_GET
END_PROPERTY

END_FUNCTION_BLOCK
